(* CODESYS project vertical_levitation_control.library
   TcLibraryId: TE140x Module Vendor|vertical_levitation_control|0.0.0.33
   Company: TE140x Module Vendor
   Title: vertical_levitation_control
   Placeholder: vertical_levitation_control
   Version: 0.0.0.33

Project tree, tasks and I/O mapping:
  POUs/
    function block FB_vertical_levitation_control [ST]: FB_exit, FB_init, nHResult, eInitExceptionHandling, eUpdateExceptionHandling, nExceptionCnt, stActiveException, bInitialized, bExecute
    TcCOM Wrapper/
      function block FB_vertical_levitation_control_TcCOM_InitStruct [ST]: FB_init, FB_afterinit, Reinit, FB_exit, eObjectState, nHResult, ipTcComObject, ipADI, nTaskOid, nTaskPriority, nTaskCycleTimeNs, nTaskPort, nTaskSortOrder, eTraceLevelMax, eModuleCaller, eCallerVerification, eStepSizeAdaptation, eExecutionSequence, bExecute, eAccessLockState, eInitExceptionHandling, eUpdateExceptionHandling, stModuleBuildInfo, bInitialized, nSkippedExecutionCount, stLibraryInfo, stModuleInfo, stModuleGeneratorInfo, stSimulinkModelInfo, evertical_levitation_control_P_Sharing, nvertical_levitation_control_P_Definer, stvertical_levitation_control_P, fSimulationTime, nCycleCount, nExceptionCount, stExceptionInfo
  DUTs/
    data type ST_FB_vertical_levitation_control_FB_Main
    data type ST_FB_vertical_levitation_control_FB_exit
    data type ST_FB_vertical_levitation_control_FB_init
    data type ST_GetSet_HRESULT
    data type E_FpExcptCtrlSetEx
    data type ST_GetSet_E_FpExcptCtrlSetEx
    data type ST_GetSet_ULINT
    data type ST_ExceptionInfo
    data type ST_GetSet_ST_ExceptionInfo
    data type ST_GetSet_BOOL
    data type T_matrix3xdouble
    data type T_matrix2xdouble
    data type T_matrix4xdouble
    data type E_SimTimeStep
    data type E_SolverMode
    data type E_ssMatrixType
    data type ST_RTWRTModelMethodsInfo
    data type E_slJmBdControl
    data type ST_ssSolverInfo
    data type T_matrix8xdouble
    data type T_matrix5xdouble
    data type T_matrix4xlogical
    data type T_matrix8xlogical
    data type ST_B_forcecurrent_BL_vertical_levitation_control_T
    data type ST_B_MATLABFunction_vertical_levitation_control_T
    data type ST_B_vertical_levitation_control_T
    data type T_ZCSigState
    data type T_matrix4xZCSigState
    data type ST_PrevZCX_vertical_levitation_control_T
    data type ST_X_vertical_levitation_control_T
    data type ST_ExtU_vertical_levitation_control_T
    data type ST_ExtY_vertical_levitation_control_T
    data type T_matrix4xbool
    data type ST_XDis_vertical_levitation_control_T
    data type T_matrix22xdouble
    data type T_matrix22x4xdouble
    data type PLREAL
    data type T_matrix4xdoublepointer
    data type ST_ODE4_IntgData
    data type ST_DW_vertical_levitation_control_T
    data type ST_x08a7a7bbd0e5d629f7d70ceec84eacfe
    data type ST_xf09845edab6c83520d8d57def6d6fe1c
    data type ST_RT_MODEL_vertical_levitation_control_T
    data type T_matrix53xdouble
    data type T_matrix1007xdouble
    data type T_matrix19xdouble
    data type T_matrix380xdouble
    data type T_matrix3xlogical
    data type ST_P_vertical_levitation_control_T
    data type E_ModuleCaller
    data type E_CallerVerification
    data type E_StepSizeAdaptation
    data type E_ExecutionSequence1
    data type E_FpExcptCtrlSet
    data type ST_TcMatSim_ModuleGeneratorInfo
    data type ST_TcMatSim_SimulinkModelInfo
    data type E_ParameterSharingType
    data type ST_FB_vertical_levitation_control_TcCOM_InitStruct
    data type ST_FB_vertical_levitation_control_TcCOM_InitStruct_FB_init
    data type ST_FB_vertical_levitation_control_TcCOM_InitStruct_FB_afterinit
    data type ST_FB_vertical_levitation_control_TcCOM_InitStruct_Reinit
    data type ST_FB_vertical_levitation_control_TcCOM_InitStruct_FB_Main
    data type ST_FB_vertical_levitation_control_TcCOM_InitStruct_FB_exit
    data type ST_GetSet_TCOM_STATE
    data type ST_GetSet_ITComObject
    data type ST_GetSet_ITcADI
    data type ST_vertical_levitation_control_U_T
    data type ST_vertical_levitation_control_Y_T
    data type ST_vertical_levitation_control_X_T
    data type ST_vertical_levitation_control_DW_T
    data type ST_GetSet_OTCID
    data type ST_GetSet_UDINT
    data type ST_GetSet_UINT
    data type ST_GetSet_TcTraceLevel
    data type ST_GetSet_E_ModuleCaller
    data type ST_GetSet_E_CallerVerification
    data type ST_GetSet_E_StepSizeAdaptation
    data type ST_GetSet_E_ExecutionSequence1
    data type ST_GetSet_E_FpExcptCtrlSet
    data type ST_ModuleBuildInfo
    data type ST_GetSet_ST_ModuleBuildInfo
    data type ST_LibraryInfo
    data type ST_GetSet_ST_LibraryInfo
    data type ST_ModuleInfo
    data type ST_GetSet_ST_ModuleInfo
    data type ST_GetSet_ST_TcMatSim_ModuleGeneratorInfo
    data type ST_GetSet_ST_TcMatSim_SimulinkModelInfo
    data type ST_GetSet_E_ParameterSharingType
    data type ST_GetSet_ST_P_vertical_levitation_control_T
    data type ST_GetSet_LREAL
  Version/
    global variables Global_Version
*)

// DUTs/ST_FB_vertical_levitation_control_FB_Main
{attribute 'TcIecLibraryType'}
{attribute 'hide'}
TYPE ST_FB_vertical_levitation_control_FB_Main : 
	STRUCT
		{attribute 'GUID' := '18071995-0000-0000-0000-000000000018'}
		pInst : PVOID;
		result : BOOL;
		 {attribute 'hide'}
		_reserved1 : UINT_24_56;
	END_STRUCT
END_TYPE

// DUTs/ST_FB_vertical_levitation_control_FB_exit
{attribute 'TcIecLibraryType'}
{attribute 'hide'}
TYPE ST_FB_vertical_levitation_control_FB_exit : 
	STRUCT
		{attribute 'GUID' := '18071995-0000-0000-0000-000000000018'}
		pInst : PVOID;
		bInCopyCode : BOOL;
		result : BOOL;
		 {attribute 'hide'}
		_reserved1 : UINT_16_48;
	END_STRUCT
END_TYPE

// DUTs/ST_FB_vertical_levitation_control_FB_init
{attribute 'TcIecLibraryType'}
{attribute 'hide'}
TYPE ST_FB_vertical_levitation_control_FB_init : 
	STRUCT
		{attribute 'GUID' := '18071995-0000-0000-0000-000000000018'}
		pInst : PVOID;
		bInitRetains : BOOL;
		bInCopyCode : BOOL;
		result : BOOL;
		 {attribute 'hide'}
		_reserved1 : UINT_8_40;
	END_STRUCT
END_TYPE

// DUTs/ST_GetSet_HRESULT
{attribute 'TcIecLibraryType'}
{attribute 'hide'}
TYPE ST_GetSet_HRESULT : 
	STRUCT
		{attribute 'GUID' := '18071995-0000-0000-0000-000000000018'}
		pInst : PVOID;
		{attribute 'GUID' := '18071995-0000-0000-0000-000000000019'}
		nParam : HRESULT;
		 {attribute 'hide'}
		_reserved1 : UINT_0_32;
	END_STRUCT
END_TYPE

// DUTs/E_FpExcptCtrlSetEx
(* Generated from type 'TcMgSdk.FpExcptCtrlSetEx' *)
{attribute 'TcIecLibraryType'}
TYPE E_FpExcptCtrlSetEx : (
	CallerExceptions:=1, 	(* Use the floating point exception settings provided by the caller *)
	ThrowExceptions:=3, 	(* Enable floating point exceptions on invalid operations and divisions by zero *)
	SuppressExceptions:=13, 	(* Disable floating point exceptions. *)
	LogExceptions:=19, 	(* Log exception information. *)
	LogAndHold:=51, 	(* Log exception information and puase execution of the cyclic code after completion of the actual cycle *)
	LogAndCatch:=83, 	(* Log exception information and immediately terminate execution of the cyclic code. Reinitialization is required to restart. *)
	LogAndDump:=147, 	(* Log exception information, create a dump file with detailed exception information and try to continue execution of the cyclic code *)
	LogHoldAndDump:=179, 	(* Log exception information, create a dump file with detailed exception information and puase execution of the cyclic code after completion of the actual cycle *)
	LogCatchAndDump:=211	(* Log exception information, create a dump file with detailed exception information and immediately terminate execution of the cyclic code. Reinitialization is required to restart. *)
) USINT;
END_TYPE

// DUTs/ST_GetSet_E_FpExcptCtrlSetEx
{attribute 'TcIecLibraryType'}
{attribute 'hide'}
TYPE ST_GetSet_E_FpExcptCtrlSetEx : 
	STRUCT
		{attribute 'GUID' := '18071995-0000-0000-0000-000000000018'}
		pInst : PVOID;
		eParam : E_FpExcptCtrlSetEx;
		 {attribute 'hide'}
		_reserved1 : UINT_24_56;
	END_STRUCT
END_TYPE

// DUTs/ST_GetSet_ULINT
{attribute 'TcIecLibraryType'}
{attribute 'hide'}
TYPE ST_GetSet_ULINT : 
	STRUCT
		{attribute 'GUID' := '18071995-0000-0000-0000-000000000018'}
		pInst : PVOID;
		nParam : ULINT;
	END_STRUCT
END_TYPE

// DUTs/ST_ExceptionInfo
(* Generated from type 'TcMgSdk.ExceptionInfo' *)
{attribute 'TcIecLibraryType'}
TYPE ST_ExceptionInfo : 
	STRUCT
		(* Generated from item 'ExceptionCode' *)
		nExceptionCode : DINT;
		(* Generated from item 'TmxName' *)
		{attribute 'GUID' := '18071995-0000-0000-0000-00010000007F'}
		sTmxName : STRING(127);
		(* Generated from item 'TmxVersion' *)
		nTmxVersion : ARRAY [0..3] OF UDINT;
		(* Generated from item 'InstructionAddr' *)
		nInstructionAddr : UDINT;
		(* Generated from item 'ReturnAddr' *)
		nReturnAddr : ARRAY [0..3] OF UDINT;
		(* Generated from item 'DumpCreated' *)
		bDumpCreated : BOOL;
		 {attribute 'hide'}
		_reserved1 : ARRAY [1..3] OF USINT;
	END_STRUCT
END_TYPE

// DUTs/ST_GetSet_ST_ExceptionInfo
{attribute 'TcIecLibraryType'}
{attribute 'hide'}
TYPE ST_GetSet_ST_ExceptionInfo : 
	STRUCT
		{attribute 'GUID' := '18071995-0000-0000-0000-000000000018'}
		pInst : PVOID;
		stParam : ST_ExceptionInfo;
		 {attribute 'hide'}
		_reserved1 : UINT_0_32;
	END_STRUCT
END_TYPE

// DUTs/ST_GetSet_BOOL
{attribute 'TcIecLibraryType'}
{attribute 'hide'}
TYPE ST_GetSet_BOOL : 
	STRUCT
		{attribute 'GUID' := '18071995-0000-0000-0000-000000000018'}
		pInst : PVOID;
		bParam : BOOL;
		 {attribute 'hide'}
		_reserved1 : UINT_24_56;
	END_STRUCT
END_TYPE

// DUTs/T_matrix3xdouble
(* Generated from type 'matrix3xdouble' *)
{attribute 'TcIecLibraryType'}
TYPE T_matrix3xdouble : ARRAY [0..2] OF LREAL;
END_TYPE

// DUTs/T_matrix2xdouble
(* Generated from type 'matrix2xdouble' *)
{attribute 'TcIecLibraryType'}
TYPE T_matrix2xdouble : ARRAY [0..1] OF LREAL;
END_TYPE

// DUTs/T_matrix4xdouble
(* Generated from type 'matrix4xdouble' *)
{attribute 'TcIecLibraryType'}
TYPE T_matrix4xdouble : ARRAY [0..3] OF LREAL;
END_TYPE

// DUTs/E_SimTimeStep
(* Generated from type 'SimTimeStep' *)
{attribute 'TcIecLibraryType'}
{attribute 'qualified_only' := 'true'}
TYPE E_SimTimeStep : (MINOR_TIME_STEP:=0, MAJOR_TIME_STEP:=1) DINT;
END_TYPE

// DUTs/E_SolverMode
(* Generated from type 'SolverMode' *)
{attribute 'TcIecLibraryType'}
{attribute 'qualified_only' := 'true'}
TYPE E_SolverMode : (SOLVER_MODE_AUTO:=0, SOLVER_MODE_SINGLETASKING:=1, SOLVER_MODE_MULTITASKING:=2) DINT;
END_TYPE

// DUTs/E_ssMatrixType
(* Generated from type 'ssMatrixType' *)
{attribute 'TcIecLibraryType'}
{attribute 'qualified_only' := 'true'}
TYPE E_ssMatrixType : (SS_MATRIX_NONE:=0, SS_MATRIX_CONSTANT:=1, SS_MATRIX_TIMEDEP:=2, SS_MATRIX_STATEDEP:=3) DINT;
END_TYPE

// DUTs/ST_RTWRTModelMethodsInfo
(* Generated from type 'RTWRTModelMethodsInfo' *)
{attribute 'TcIecLibraryType'}
TYPE ST_RTWRTModelMethodsInfo : 
	STRUCT
		(* Generated from item 'rtModelPtr' *)
		{attribute 'GUID' := '18071995-0000-0000-0000-000000000018'}
		prtModelPtr : PVOID;
		(* Generated from item 'rtmInitSizesFcn' *)
		{attribute 'GUID' := '18071995-0000-0000-0000-000000000018'}
		prtmInitSizesFcn : PVOID;
		(* Generated from item 'rtmInitSampTimesFcn' *)
		{attribute 'GUID' := '18071995-0000-0000-0000-000000000018'}
		prtmInitSampTimesFcn : PVOID;
		(* Generated from item 'rtmStartFcn' *)
		{attribute 'GUID' := '18071995-0000-0000-0000-000000000018'}
		prtmStartFcn : PVOID;
		(* Generated from item 'rtmOutputsFcn' *)
		{attribute 'GUID' := '18071995-0000-0000-0000-000000000018'}
		prtmOutputsFcn : PVOID;
		(* Generated from item 'rtmUpdateFcn' *)
		{attribute 'GUID' := '18071995-0000-0000-0000-000000000018'}
		prtmUpdateFcn : PVOID;
		(* Generated from item 'rtmDervisFcn' *)
		{attribute 'GUID' := '18071995-0000-0000-0000-000000000018'}
		prtmDervisFcn : PVOID;
		(* Generated from item 'rtmProjectionFcn' *)
		{attribute 'GUID' := '18071995-0000-0000-0000-000000000018'}
		prtmProjectionFcn : PVOID;
		(* Generated from item 'rtmMassMatrixFcn' *)
		{attribute 'GUID' := '18071995-0000-0000-0000-000000000018'}
		prtmMassMatrixFcn : PVOID;
		(* Generated from item 'rtmForcingFunctionFcn' *)
		{attribute 'GUID' := '18071995-0000-0000-0000-000000000018'}
		prtmForcingFunctionFcn : PVOID;
		(* Generated from item 'rtmTerminateFcn' *)
		{attribute 'GUID' := '18071995-0000-0000-0000-000000000018'}
		prtmTerminateFcn : PVOID;
		(* Generated from item 'rtmDiscreteEventsFcn' *)
		{attribute 'GUID' := '18071995-0000-0000-0000-000000000018'}
		prtmDiscreteEventsFcn : PVOID;
	END_STRUCT
END_TYPE

// DUTs/E_slJmBdControl
(* Generated from type 'slJmBdControl' *)
{attribute 'TcIecLibraryType'}
{attribute 'qualified_only' := 'true'}
TYPE E_slJmBdControl : (SL_JM_BD_AUTO:=0, SL_JM_BD_SPARSE_PERTURBATION:=1, SL_JM_BD_FULL_PERTURBATION:=2, SL_JM_BD_SPARSE_ANALYTICAL:=3, SL_JM_BD_FULL_ANALYTICAL:=4) DINT;
END_TYPE

// DUTs/ST_ssSolverInfo
(* Generated from type 'ssSolverInfo' *)
{attribute 'TcIecLibraryType'}
TYPE ST_ssSolverInfo : 
	STRUCT
		(* Generated from item 'rtModelPtr' *)
		{attribute 'GUID' := '18071995-0000-0000-0000-000000000018'}
		prtModelPtr : PVOID;
		simTimeStepPtr : POINTER TO E_SimTimeStep;
		(* Generated from item 'solverData' *)
		{attribute 'GUID' := '18071995-0000-0000-0000-000000000018'}
		psolverData : PVOID;
		solverName : POINTER TO SINT;
		(* Generated from item 'isVariableStepSolver' *)
		bisVariableStepSolver : BOOL;
		(* Generated from item 'solverNeedsReset' *)
		bsolverNeedsReset : BOOL;
		 {attribute 'hide'}
		_reserved1 : UINT;
		(* Generated from item 'solverMode' *)
		esolverMode : E_SolverMode;
		(* Generated from item 'solverStopTime' *)
		fsolverStopTime : LREAL;
		stepSizePtr : POINTER TO LREAL;
		(* Generated from item 'minStepSize' *)
		fminStepSize : LREAL;
		(* Generated from item 'maxStepSize' *)
		fmaxStepSize : LREAL;
		(* Generated from item 'fixedStepSize' *)
		ffixedStepSize : LREAL;
		(* Generated from item 'solverShapePreserveControl' *)
		nsolverShapePreserveControl : DINT;
		(* Generated from item 'solverMaxConsecutiveMinStep' *)
		nsolverMaxConsecutiveMinStep : DINT;
		(* Generated from item 'maxNumMinSteps' *)
		nmaxNumMinSteps : DINT;
		(* Generated from item 'solverMaxOrder' *)
		nsolverMaxOrder : DINT;
		(* Generated from item 'solverConsecutiveZCsStepRelTol' *)
		fsolverConsecutiveZCsStepRelTol : LREAL;
		(* Generated from item 'solverMaxConsecutiveZCs' *)
		nsolverMaxConsecutiveZCs : DINT;
		(* Generated from item 'solverExtrapolationOrder' *)
		nsolverExtrapolationOrder : DINT;
		(* Generated from item 'solverNumberNewtonIterations' *)
		nsolverNumberNewtonIterations : DINT;
		(* Generated from item 'solverRefineFactor' *)
		nsolverRefineFactor : DINT;
		(* Generated from item 'solverRelTol' *)
		fsolverRelTol : LREAL;
		(* Generated from item 'unused_real_T_1' *)
		funused_real_T_1 : LREAL;
		dXPtr : POINTER TO POINTER TO LREAL;
		tPtr : POINTER TO POINTER TO LREAL;
		numContStatesPtr : POINTER TO DINT;
		contStatesPtr : POINTER TO POINTER TO LREAL;
		numPeriodicContStatesPtr : POINTER TO DINT;
		periodicContStateIndicesPtr : POINTER TO POINTER TO DINT;
		periodicContStateRangesPtr : POINTER TO POINTER TO LREAL;
		zcSignalVector : POINTER TO LREAL;
		zcEventsVector : POINTER TO USINT;
		zcSignalAttrib : POINTER TO USINT;
		(* Generated from item 'zcSignalVectorLength' *)
		nzcSignalVectorLength : DINT;
		 {attribute 'hide'}
		_reserved2 : UINT_0_32;
		reserved : POINTER TO USINT;
		(* Generated from item 'foundContZcEvents' *)
		bfoundContZcEvents : BOOL;
		(* Generated from item 'isAtLeftPostOfContZcEvent' *)
		bisAtLeftPostOfContZcEvent : BOOL;
		(* Generated from item 'isAtRightPostOfContZcEvent' *)
		bisAtRightPostOfContZcEvent : BOOL;
		(* Generated from item 'adaptiveZcDetection' *)
		badaptiveZcDetection : BOOL;
		(* Generated from item 'numZcSignals' *)
		nnumZcSignals : DINT;
		(* Generated from item 'stateProjection' *)
		bstateProjection : BOOL;
		(* Generated from item 'robustResetMethod' *)
		brobustResetMethod : BOOL;
		(* Generated from item 'updateJacobianAtReset' *)
		bupdateJacobianAtReset : BOOL;
		(* Generated from item 'consistencyChecking' *)
		bconsistencyChecking : BOOL;
		(* Generated from item 'massMatrixType' *)
		emassMatrixType : E_ssMatrixType;
		(* Generated from item 'massMatrixNzMax' *)
		nmassMatrixNzMax : DINT;
		 {attribute 'hide'}
		_reserved3 : UINT_0_32;
		massMatrixIr : POINTER TO DINT;
		massMatrixJc : POINTER TO DINT;
		massMatrixPr : POINTER TO LREAL;
		errStatusPtr : POINTER TO POINTER TO SINT;
		modelMethodsPtr : POINTER TO ST_RTWRTModelMethodsInfo;
		(* Generated from item 'zcThreshold' *)
		fzcThreshold : LREAL;
		(* Generated from item 'reserved_1' *)
		nreserved_1 : DINT;
		(* Generated from item 'consecutiveZCsError' *)
		nconsecutiveZCsError : DINT;
		(* Generated from item 'CTOutputIncnstWithState' *)
		bCTOutputIncnstWithState : BOOL;
		(* Generated from item 'isComputingJacobian' *)
		bisComputingJacobian : BOOL;
		 {attribute 'hide'}
		_reserved4 : UINT;
		(* Generated from item 'solverJacobianMethodControl' *)
		esolverJacobianMethodControl : E_slJmBdControl;
		(* Generated from item 'ignoredZcDiagnostic' *)
		nignoredZcDiagnostic : DINT;
		(* Generated from item 'maskedZcDiagnostic' *)
		nmaskedZcDiagnostic : DINT;
		(* Generated from item 'isOutputMethodComputed' *)
		bisOutputMethodComputed : BOOL;
		 {attribute 'hide'}
		_reserved5 : ARRAY [1..3] OF USINT;
		(* Generated from item 'maxZcBracketingIterations' *)
		nmaxZcBracketingIterations : DINT;
		(* Generated from item 'isMinorTimeStepWithModeChange' *)
		bisMinorTimeStepWithModeChange : BOOL;
		 {attribute 'hide'}
		_reserved6 : ARRAY [1..3] OF USINT;
		(* Generated from item 'maxZcPerStep' *)
		nmaxZcPerStep : DINT;
		zcSignalPtr : POINTER TO POINTER TO LREAL;
		(* Generated from item 'contStateDisabledPtr' *)
		bcontStateDisabledPtr : POINTER TO POINTER TO BOOL;
		(* Generated from item 'isContModeFrozen' *)
		bisContModeFrozen : BOOL;
		 {attribute 'hide'}
		_reserved7 : ARRAY [1..7] OF USINT;
	END_STRUCT
END_TYPE

// DUTs/T_matrix8xdouble
(* Generated from type 'matrix8xdouble' *)
{attribute 'TcIecLibraryType'}
TYPE T_matrix8xdouble : ARRAY [0..7] OF LREAL;
END_TYPE

// DUTs/T_matrix5xdouble
(* Generated from type 'matrix5xdouble' *)
{attribute 'TcIecLibraryType'}
TYPE T_matrix5xdouble : ARRAY [0..4] OF LREAL;
END_TYPE

// DUTs/T_matrix4xlogical
(* Generated from type 'matrix4xlogical' *)
{attribute 'TcIecLibraryType'}
{attribute 'BaseTypeGUID' := '18071995-0000-0000-0000-000000000030'}
TYPE T_matrix4xlogical : ARRAY [0..3] OF BOOL;
END_TYPE

// DUTs/T_matrix8xlogical
(* Generated from type 'matrix8xlogical' *)
{attribute 'TcIecLibraryType'}
{attribute 'BaseTypeGUID' := '18071995-0000-0000-0000-000000000030'}
TYPE T_matrix8xlogical : ARRAY [0..7] OF BOOL;
END_TYPE

// DUTs/ST_B_forcecurrent_BL_vertical_levitation_control_T
(* Generated from type 'B_forcecurrent_BL_vertical_levitation_control_T' *)
{attribute 'TcIecLibraryType'}
TYPE ST_B_forcecurrent_BL_vertical_levitation_control_T : 
	STRUCT
		(* Generated from item 'current_reqf' *)
		fcurrent_reqf : LREAL;
		(* Generated from item 'current_reqb' *)
		fcurrent_reqb : LREAL;
	END_STRUCT
END_TYPE

// DUTs/ST_B_MATLABFunction_vertical_levitation_control_T
(* Generated from type 'B_MATLABFunction_vertical_levitation_control_T' *)
{attribute 'TcIecLibraryType'}
TYPE ST_B_MATLABFunction_vertical_levitation_control_T : 
	STRUCT
		(* Generated from item 'y' *)
		ay : T_matrix8xdouble;
	END_STRUCT
END_TYPE

// DUTs/ST_B_vertical_levitation_control_T
(* Generated from type 'B_vertical_levitation_control_T' *)
{attribute 'TcIecLibraryType'}
TYPE ST_B_vertical_levitation_control_T : 
	STRUCT
		(* Generated from item 'UnitDelay' *)
		aUnitDelay : T_matrix4xdouble;
		(* Generated from item 'Switch1' *)
		aSwitch1 : T_matrix4xdouble;
		(* Generated from item 'Switch1_d' *)
		aSwitch1_d : T_matrix4xdouble;
		(* Generated from item 'Gain3' *)
		fGain3 : LREAL;
		(* Generated from item 'Gain7' *)
		fGain7 : LREAL;
		(* Generated from item 'Switch2' *)
		aSwitch2 : T_matrix4xdouble;
		(* Generated from item 'select_maxs' *)
		aselect_maxs : T_matrix4xdouble;
		(* Generated from item 'Delay' *)
		aDelay : T_matrix3xdouble;
		(* Generated from item 'UnitDelay1' *)
		fUnitDelay1 : LREAL;
		(* Generated from item 'FilterCoefficient' *)
		fFilterCoefficient : LREAL;
		(* Generated from item 'Saturation' *)
		fSaturation : LREAL;
		(* Generated from item 'error_integrator' *)
		ferror_integrator : LREAL;
		(* Generated from item 'Gain10' *)
		fGain10 : LREAL;
		(* Generated from item 'Integrator' *)
		fIntegrator : LREAL;
		(* Generated from item 'Filtertotgain' *)
		fFiltertotgain : LREAL;
		(* Generated from item 'Add4' *)
		fAdd4 : LREAL;
		(* Generated from item 'UnitDelay1_g' *)
		fUnitDelay1_g : LREAL;
		(* Generated from item 'Sum' *)
		fSum : LREAL;
		(* Generated from item 'Gain12' *)
		fGain12 : LREAL;
		(* Generated from item 'Integrator_g' *)
		fIntegrator_g : LREAL;
		(* Generated from item 'K_D_roll' *)
		fK_D_roll : LREAL;
		(* Generated from item 'Filterrollgain' *)
		fFilterrollgain : LREAL;
		(* Generated from item 'TSamp' *)
		fTSamp : LREAL;
		(* Generated from item 'Diff' *)
		fDiff : LREAL;
		(* Generated from item 'Add4_g' *)
		fAdd4_g : LREAL;
		(* Generated from item 'UnitDelay1_i' *)
		fUnitDelay1_i : LREAL;
		(* Generated from item 'Add4_gu' *)
		fAdd4_gu : LREAL;
		(* Generated from item 'UnitDelay1_d' *)
		fUnitDelay1_d : LREAL;
		(* Generated from item 'Switch' *)
		fSwitch : LREAL;
		(* Generated from item 'Gain13' *)
		fGain13 : LREAL;
		(* Generated from item 'Integrator_i' *)
		fIntegrator_i : LREAL;
		(* Generated from item 'Filterpitgain' *)
		fFilterpitgain : LREAL;
		(* Generated from item 'Add4_l' *)
		fAdd4_l : LREAL;
		(* Generated from item 'UnitDelay1_e' *)
		fUnitDelay1_e : LREAL;
		(* Generated from item 'Sum_j' *)
		fSum_j : LREAL;
		(* Generated from item 'select_mins' *)
		aselect_mins : T_matrix4xdouble;
		(* Generated from item 'Switch_i' *)
		fSwitch_i : LREAL;
		(* Generated from item 'UnitDelay1_m' *)
		fUnitDelay1_m : LREAL;
		(* Generated from item 'FilterCoefficient_l' *)
		fFilterCoefficient_l : LREAL;
		(* Generated from item 'Saturation_p' *)
		fSaturation_p : LREAL;
		(* Generated from item 'Switch1_a' *)
		fSwitch1_a : LREAL;
		(* Generated from item 'UnitDelay1_n' *)
		fUnitDelay1_n : LREAL;
		(* Generated from item 'FilterCoefficient_o' *)
		fFilterCoefficient_o : LREAL;
		(* Generated from item 'Saturation_pi' *)
		fSaturation_pi : LREAL;
		(* Generated from item 'Switch2_j' *)
		fSwitch2_j : LREAL;
		(* Generated from item 'F_hemsfinal' *)
		aF_hemsfinal : T_matrix4xdouble;
		(* Generated from item 'Switch2_f' *)
		aSwitch2_f : T_matrix8xdouble;
		(* Generated from item 'Switch_o' *)
		fSwitch_o : LREAL;
		(* Generated from item 'Switch_j' *)
		fSwitch_j : LREAL;
		(* Generated from item 'Switch_k' *)
		fSwitch_k : LREAL;
		(* Generated from item 'Divide' *)
		fDivide : LREAL;
		(* Generated from item 'Add5' *)
		fAdd5 : LREAL;
		(* Generated from item 'Add6' *)
		fAdd6 : LREAL;
		(* Generated from item 'Gain' *)
		fGain : LREAL;
		(* Generated from item 'UnitDelay2' *)
		fUnitDelay2 : LREAL;
		(* Generated from item 'Sum4' *)
		fSum4 : LREAL;
		(* Generated from item 'Sum5' *)
		fSum5 : LREAL;
		(* Generated from item 'Add5_p' *)
		fAdd5_p : LREAL;
		(* Generated from item 'Add6_l' *)
		fAdd6_l : LREAL;
		(* Generated from item 'Gain_m' *)
		fGain_m : LREAL;
		(* Generated from item 'UnitDelay2_i' *)
		fUnitDelay2_i : LREAL;
		(* Generated from item 'Sum4_d' *)
		fSum4_d : LREAL;
		(* Generated from item 'Sum5_m' *)
		fSum5_m : LREAL;
		(* Generated from item 'Add5_f' *)
		fAdd5_f : LREAL;
		(* Generated from item 'Add6_a' *)
		fAdd6_a : LREAL;
		(* Generated from item 'Gain_j' *)
		fGain_j : LREAL;
		(* Generated from item 'UnitDelay2_m' *)
		fUnitDelay2_m : LREAL;
		(* Generated from item 'Sum4_g' *)
		fSum4_g : LREAL;
		(* Generated from item 'Sum5_g' *)
		fSum5_g : LREAL;
		(* Generated from item 'Add5_h' *)
		fAdd5_h : LREAL;
		(* Generated from item 'Add6_h' *)
		fAdd6_h : LREAL;
		(* Generated from item 'Gain_l' *)
		fGain_l : LREAL;
		(* Generated from item 'UnitDelay2_o' *)
		fUnitDelay2_o : LREAL;
		(* Generated from item 'Sum4_i' *)
		fSum4_i : LREAL;
		(* Generated from item 'Sum5_j' *)
		fSum5_j : LREAL;
		(* Generated from item 'IsPeak1' *)
		aIsPeak1 : T_matrix4xdouble;
		(* Generated from item 'Switch2_d' *)
		aSwitch2_d : T_matrix4xdouble;
		(* Generated from item 'F_netpostfm' *)
		aF_netpostfm : T_matrix3xdouble;
		(* Generated from item 'clamppit' *)
		fclamppit : LREAL;
		(* Generated from item 'clamproll' *)
		fclamproll : LREAL;
		(* Generated from item 'clamptot' *)
		fclamptot : LREAL;
		(* Generated from item 'K_I_tot' *)
		fK_I_tot : LREAL;
		(* Generated from item 'K_I_roll' *)
		fK_I_roll : LREAL;
		(* Generated from item 'K_I_pit' *)
		fK_I_pit : LREAL;
		(* Generated from item 'current_reqf' *)
		fcurrent_reqf : LREAL;
		(* Generated from item 'current_reqb' *)
		fcurrent_reqb : LREAL;
		(* Generated from item 'current_reqf_c' *)
		fcurrent_reqf_c : LREAL;
		(* Generated from item 'current_reqb_c' *)
		fcurrent_reqb_c : LREAL;
		(* Generated from item 'F_hems' *)
		aF_hems : T_matrix4xdouble;
		(* Generated from item 'Switch2_l' *)
		aSwitch2_l : T_matrix4xdouble;
		(* Generated from item 'Sum5_f' *)
		fSum5_f : LREAL;
		(* Generated from item 'Is' *)
		aIs : T_matrix4xdouble;
		(* Generated from item 'satn' *)
		asatn : T_matrix8xdouble;
		(* Generated from item 'airgaps_avg' *)
		aairgaps_avg : T_matrix4xdouble;
		(* Generated from item 'airgap_diff' *)
		fairgap_diff : LREAL;
		(* Generated from item 'tau_x' *)
		ftau_x : LREAL;
		(* Generated from item 'Sum_l' *)
		fSum_l : LREAL;
		(* Generated from item 'corrected_out' *)
		fcorrected_out : LREAL;
		(* Generated from item 'corrected_out_j' *)
		fcorrected_out_j : LREAL;
		(* Generated from item 'corrected_out_o' *)
		fcorrected_out_o : LREAL;
		(* Generated from item 'F_hems_b' *)
		aF_hems_b : T_matrix4xdouble;
		(* Generated from item 'clamp_tot' *)
		aclamp_tot : T_matrix2xdouble;
		(* Generated from item 'clamp_roll' *)
		aclamp_roll : T_matrix2xdouble;
		(* Generated from item 'clamp_pit' *)
		aclamp_pit : T_matrix2xdouble;
		(* Generated from item 'counter' *)
		acounter : T_matrix5xdouble;
		(* Generated from item 'F_dof_sat' *)
		aF_dof_sat : T_matrix3xdouble;
		(* Generated from item 'sat_fail' *)
		fsat_fail : LREAL;
		(* Generated from item 'q' *)
		fq : LREAL;
		(* Generated from item 'q_m' *)
		fq_m : LREAL;
		(* Generated from item 'q_f' *)
		fq_f : LREAL;
		(* Generated from item 'q_d' *)
		fq_d : LREAL;
		(* Generated from item 'UnaryMinus' *)
		fUnaryMinus : LREAL;
		(* Generated from item 'UnaryMinus_b' *)
		fUnaryMinus_b : LREAL;
		(* Generated from item 'UnaryMinus_n' *)
		fUnaryMinus_n : LREAL;
		(* Generated from item 'UnaryMinus_l' *)
		fUnaryMinus_l : LREAL;
		(* Generated from item 'Integrator2' *)
		aIntegrator2 : T_matrix4xdouble;
		(* Generated from item 'Switch_ka' *)
		aSwitch_ka : T_matrix4xdouble;
		(* Generated from item 'K_P_tot' *)
		fK_P_tot : LREAL;
		(* Generated from item 'Product1' *)
		fProduct1 : LREAL;
		(* Generated from item 'Product1_p' *)
		fProduct1_p : LREAL;
		(* Generated from item 'Product1_i' *)
		fProduct1_i : LREAL;
		(* Generated from item 'TmpSignalConversionAtSFunctionInport1' *)
		aTmpSignalConversionAtSFunctionInport1 : T_matrix3xdouble;
		(* Generated from item 't' *)
		ft : LREAL;
		(* Generated from item 's' *)
		fs : LREAL;
		(* Generated from item 'v' *)
		fv : LREAL;
		(* Generated from item 't_m' *)
		ft_m : LREAL;
		(* Generated from item 's_b' *)
		fs_b : LREAL;
		(* Generated from item 'v_i' *)
		fv_i : LREAL;
		(* Generated from item 't_k' *)
		ft_k : LREAL;
		(* Generated from item 's_i' *)
		fs_i : LREAL;
		(* Generated from item 'v_l' *)
		fv_l : LREAL;
		(* Generated from item 't_i' *)
		ft_i : LREAL;
		(* Generated from item 's_iy' *)
		fs_iy : LREAL;
		(* Generated from item 'v_if' *)
		fv_if : LREAL;
		(* Generated from item 'Integrator_f' *)
		fIntegrator_f : LREAL;
		(* Generated from item 'Switch_h' *)
		fSwitch_h : LREAL;
		(* Generated from item 'u' *)
		fu : LREAL;
		(* Generated from item 'u_h' *)
		fu_h : LREAL;
		(* Generated from item 'u_ha' *)
		fu_ha : LREAL;
		(* Generated from item 'Final_ON' *)
		aFinal_ON : T_matrix8xdouble;
		(* Generated from item 'Abs1' *)
		aAbs1 : T_matrix4xdouble;
		(* Generated from item 'IntegralGain' *)
		fIntegralGain : LREAL;
		(* Generated from item 'u_f' *)
		fu_f : LREAL;
		(* Generated from item 'IntegralGain_e' *)
		fIntegralGain_e : LREAL;
		(* Generated from item 'SignPreSat' *)
		fSignPreSat : LREAL;
		(* Generated from item 'IntegralGain_h' *)
		fIntegralGain_h : LREAL;
		(* Generated from item 'Product4' *)
		fProduct4 : LREAL;
		(* Generated from item 'Product4_b' *)
		fProduct4_b : LREAL;
		(* Generated from item 'Product4_e' *)
		fProduct4_e : LREAL;
		(* Generated from item 'Product4_d' *)
		fProduct4_d : LREAL;
		(* Generated from item 'Product3' *)
		fProduct3 : LREAL;
		(* Generated from item 'SignPreSat_g' *)
		fSignPreSat_g : LREAL;
		(* Generated from item 'SignPreSat_b' *)
		fSignPreSat_b : LREAL;
		(* Generated from item 'Product4_a' *)
		fProduct4_a : LREAL;
		(* Generated from item 'Sign' *)
		fSign : LREAL;
		(* Generated from item 'Sign1' *)
		fSign1 : LREAL;
		(* Generated from item 'Delay1' *)
		fDelay1 : REAL;
		(* Generated from item 'fmsatfailordisabled' *)
		ffmsatfailordisabled : REAL;
		(* Generated from item 'hard_disable_fmm' *)
		fhard_disable_fmm : REAL;
		(* Generated from item 'enabled' *)
		nenabled : USINT;
		(* Generated from item 'DataTypeConv2' *)
		nDataTypeConv2 : SINT;
		(* Generated from item 'DataTypeConv1' *)
		nDataTypeConv1 : SINT;
		(* Generated from item 'didfmcausesattofail' *)
		adidfmcausesattofail : T_matrix4xlogical;
		(* Generated from item 'AND3' *)
		bAND3 : BOOL;
		(* Generated from item 'Memory' *)
		bMemory : BOOL;
		(* Generated from item 'AND3_d' *)
		bAND3_d : BOOL;
		(* Generated from item 'Memory_p' *)
		bMemory_p : BOOL;
		(* Generated from item 'AND3_l' *)
		bAND3_l : BOOL;
		(* Generated from item 'Memory_f' *)
		bMemory_f : BOOL;
		(* Generated from item 'y' *)
		_by : BOOL;
		(* Generated from item 'LowerRelop1' *)
		aLowerRelop1 : T_matrix4xlogical;
		(* Generated from item 'UpperRelop' *)
		aUpperRelop : T_matrix4xlogical;
		(* Generated from item 'LowerRelop1_c' *)
		aLowerRelop1_c : T_matrix8xlogical;
		(* Generated from item 'UpperRelop_o' *)
		aUpperRelop_o : T_matrix8xlogical;
		(* Generated from item 'LowerRelop1_e' *)
		aLowerRelop1_e : T_matrix4xlogical;
		(* Generated from item 'CastToBoolean' *)
		bCastToBoolean : BOOL;
		(* Generated from item 'AND' *)
		bAND : BOOL;
		(* Generated from item 'sf_forcecurrent_FR' *)
		stsf_forcecurrent_FR : ST_B_forcecurrent_BL_vertical_levitation_control_T;
		(* Generated from item 'sf_forcecurrent_BL' *)
		stsf_forcecurrent_BL : ST_B_forcecurrent_BL_vertical_levitation_control_T;
		(* Generated from item 'sf_MATLABFunction1' *)
		stsf_MATLABFunction1 : ST_B_MATLABFunction_vertical_levitation_control_T;
		(* Generated from item 'sf_MATLABFunction' *)
		stsf_MATLABFunction : ST_B_MATLABFunction_vertical_levitation_control_T;
	END_STRUCT
END_TYPE

// DUTs/T_ZCSigState
(* Generated from type 'ZCSigState' *)
{attribute 'TcIecLibraryType'}
TYPE T_ZCSigState : USINT;
END_TYPE

// DUTs/T_matrix4xZCSigState
(* Generated from type 'matrix4xZCSigState' *)
{attribute 'TcIecLibraryType'}
{attribute 'BaseTypeGUID' := 'CF0EC509-8CFA-173E-6D32-2A6837BC8565'}
TYPE T_matrix4xZCSigState : ARRAY [0..3] OF T_ZCSigState;
END_TYPE

// DUTs/ST_PrevZCX_vertical_levitation_control_T
(* Generated from type 'PrevZCX_vertical_levitation_control_T' *)
{attribute 'TcIecLibraryType'}
TYPE ST_PrevZCX_vertical_levitation_control_T : 
	STRUCT
		(* Generated from item 'Integrator1_Reset_ZCE' *)
		aIntegrator1_Reset_ZCE : T_matrix4xZCSigState;
		(* Generated from item 'Integrator_Reset_ZCE' *)
		nIntegrator_Reset_ZCE : T_ZCSigState;
		(* Generated from item 'Filter_Reset_ZCE' *)
		nFilter_Reset_ZCE : T_ZCSigState;
		(* Generated from item 'error_integrator_Reset_ZCE' *)
		nerror_integrator_Reset_ZCE : T_ZCSigState;
		(* Generated from item 'time_integrator_Reset_ZCE' *)
		ntime_integrator_Reset_ZCE : T_ZCSigState;
		(* Generated from item 'Integrator_Reset_ZCE_k' *)
		nIntegrator_Reset_ZCE_k : T_ZCSigState;
		(* Generated from item 'Filtertot_Reset_ZCE' *)
		nFiltertot_Reset_ZCE : T_ZCSigState;
		(* Generated from item 'Integrator_Reset_ZCE_m' *)
		nIntegrator_Reset_ZCE_m : T_ZCSigState;
		(* Generated from item 'Filterroll_Reset_ZCE' *)
		nFilterroll_Reset_ZCE : T_ZCSigState;
		(* Generated from item 'Integrator_Reset_ZCE_km' *)
		nIntegrator_Reset_ZCE_km : T_ZCSigState;
		(* Generated from item 'Filterpit_Reset_ZCE' *)
		nFilterpit_Reset_ZCE : T_ZCSigState;
		(* Generated from item 'Integrator_Reset_ZCE_b' *)
		nIntegrator_Reset_ZCE_b : T_ZCSigState;
		(* Generated from item 'Filter_Reset_ZCE_m' *)
		nFilter_Reset_ZCE_m : T_ZCSigState;
		(* Generated from item 'Integrator_Reset_ZCE_d' *)
		nIntegrator_Reset_ZCE_d : T_ZCSigState;
		(* Generated from item 'Filter_Reset_ZCE_a' *)
		nFilter_Reset_ZCE_a : T_ZCSigState;
		(* Generated from item 'Integrator2_Reset_ZCE' *)
		aIntegrator2_Reset_ZCE : T_matrix4xZCSigState;
	END_STRUCT
END_TYPE

// DUTs/ST_X_vertical_levitation_control_T
(* Generated from type 'X_vertical_levitation_control_T' *)
{attribute 'TcIecLibraryType'}
TYPE ST_X_vertical_levitation_control_T : 
	STRUCT
		(* Generated from item 'Integrator1_CSTATE' *)
		aIntegrator1_CSTATE : T_matrix4xdouble;
		(* Generated from item 'Integrator_CSTATE' *)
		fIntegrator_CSTATE : LREAL;
		(* Generated from item 'Filter_CSTATE' *)
		fFilter_CSTATE : LREAL;
		(* Generated from item 'error_integrator_CSTATE' *)
		ferror_integrator_CSTATE : LREAL;
		(* Generated from item 'time_integrator_CSTATE' *)
		ftime_integrator_CSTATE : LREAL;
		(* Generated from item 'Integrator_CSTATE_p' *)
		fIntegrator_CSTATE_p : LREAL;
		(* Generated from item 'Filtertot_CSTATE' *)
		fFiltertot_CSTATE : LREAL;
		(* Generated from item 'Integrator_CSTATE_k' *)
		fIntegrator_CSTATE_k : LREAL;
		(* Generated from item 'Filterroll_CSTATE' *)
		fFilterroll_CSTATE : LREAL;
		(* Generated from item 'Integrator_CSTATE_pl' *)
		fIntegrator_CSTATE_pl : LREAL;
		(* Generated from item 'Filterpit_CSTATE' *)
		fFilterpit_CSTATE : LREAL;
		(* Generated from item 'Integrator_CSTATE_c' *)
		fIntegrator_CSTATE_c : LREAL;
		(* Generated from item 'Filter_CSTATE_j' *)
		fFilter_CSTATE_j : LREAL;
		(* Generated from item 'Integrator_CSTATE_pq' *)
		fIntegrator_CSTATE_pq : LREAL;
		(* Generated from item 'Filter_CSTATE_b' *)
		fFilter_CSTATE_b : LREAL;
		(* Generated from item 'Integrator2_CSTATE' *)
		aIntegrator2_CSTATE : T_matrix4xdouble;
	END_STRUCT
END_TYPE

// DUTs/ST_ExtU_vertical_levitation_control_T
(* Generated from type 'ExtU_vertical_levitation_control_T' *)
{attribute 'TcIecLibraryType'}
TYPE ST_ExtU_vertical_levitation_control_T : 
	STRUCT
		(* Generated from item 'z_avg' *)
		fz_avg : LREAL;
		(* Generated from item 'roll_measured' *)
		froll_measured : LREAL;
		(* Generated from item 'pitch_measured' *)
		fpitch_measured : LREAL;
		(* Generated from item 'ems_roll' *)
		fems_roll : LREAL;
		(* Generated from item 'F_imu' *)
		aF_imu : T_matrix3xdouble;
		(* Generated from item 'gyro_imu' *)
		agyro_imu : T_matrix3xdouble;
		(* Generated from item 'motor_Fy_l' *)
		fmotor_Fy_l : LREAL;
		(* Generated from item 'motor_Fy_r' *)
		fmotor_Fy_r : LREAL;
		(* Generated from item 'Feedback_current_hems' *)
		fFeedback_current_hems : LREAL;
	END_STRUCT
END_TYPE

// DUTs/ST_ExtY_vertical_levitation_control_T
(* Generated from type 'ExtY_vertical_levitation_control_T' *)
{attribute 'TcIecLibraryType'}
TYPE ST_ExtY_vertical_levitation_control_T : 
	STRUCT
		(* Generated from item 'I_VFL' *)
		aI_VFL : T_matrix2xdouble;
		(* Generated from item 'I_VFR' *)
		aI_VFR : T_matrix2xdouble;
		(* Generated from item 'I_VBL' *)
		aI_VBL : T_matrix2xdouble;
		(* Generated from item 'I_VBR' *)
		aI_VBR : T_matrix2xdouble;
		(* Generated from item 'F_hems' *)
		aF_hems : T_matrix4xdouble;
		(* Generated from item 'F_requested' *)
		aF_requested : T_matrix3xdouble;
		(* Generated from item 'integral_terms' *)
		aintegral_terms : T_matrix3xdouble;
		(* Generated from item 'sat_failed' *)
		fsat_failed : LREAL;
		(* Generated from item 'net_post_sat' *)
		anet_post_sat : T_matrix3xdouble;
		(* Generated from item 'z_target_adjusted' *)
		fz_target_adjusted : LREAL;
		(* Generated from item 'Max_allowed_current' *)
		aMax_allowed_current : T_matrix4xdouble;
		(* Generated from item 'Min_allowed_current' *)
		aMin_allowed_current : T_matrix4xdouble;
		(* Generated from item 'Avg_total_hems_current' *)
		fAvg_total_hems_current : LREAL;
		(* Generated from item 'Avg_current_hems' *)
		fAvg_current_hems : LREAL;
	END_STRUCT
END_TYPE

// DUTs/T_matrix4xbool
(* Generated from type 'matrix4xbool' *)
{attribute 'TcIecLibraryType'}
{attribute 'BaseTypeGUID' := '18071995-0000-0000-0000-000000000030'}
TYPE T_matrix4xbool : ARRAY [0..3] OF BOOL;
END_TYPE

// DUTs/ST_XDis_vertical_levitation_control_T
(* Generated from type 'XDis_vertical_levitation_control_T' *)
{attribute 'TcIecLibraryType'}
TYPE ST_XDis_vertical_levitation_control_T : 
	STRUCT
		(* Generated from item 'Integrator1_CSTATE' *)
		aIntegrator1_CSTATE : T_matrix4xbool;
		(* Generated from item 'Integrator_CSTATE' *)
		bIntegrator_CSTATE : BOOL;
		(* Generated from item 'Filter_CSTATE' *)
		bFilter_CSTATE : BOOL;
		(* Generated from item 'error_integrator_CSTATE' *)
		berror_integrator_CSTATE : BOOL;
		(* Generated from item 'time_integrator_CSTATE' *)
		btime_integrator_CSTATE : BOOL;
		(* Generated from item 'Integrator_CSTATE_p' *)
		bIntegrator_CSTATE_p : BOOL;
		(* Generated from item 'Filtertot_CSTATE' *)
		bFiltertot_CSTATE : BOOL;
		(* Generated from item 'Integrator_CSTATE_k' *)
		bIntegrator_CSTATE_k : BOOL;
		(* Generated from item 'Filterroll_CSTATE' *)
		bFilterroll_CSTATE : BOOL;
		(* Generated from item 'Integrator_CSTATE_pl' *)
		bIntegrator_CSTATE_pl : BOOL;
		(* Generated from item 'Filterpit_CSTATE' *)
		bFilterpit_CSTATE : BOOL;
		(* Generated from item 'Integrator_CSTATE_c' *)
		bIntegrator_CSTATE_c : BOOL;
		(* Generated from item 'Filter_CSTATE_j' *)
		bFilter_CSTATE_j : BOOL;
		(* Generated from item 'Integrator_CSTATE_pq' *)
		bIntegrator_CSTATE_pq : BOOL;
		(* Generated from item 'Filter_CSTATE_b' *)
		bFilter_CSTATE_b : BOOL;
		(* Generated from item 'Integrator2_CSTATE' *)
		aIntegrator2_CSTATE : T_matrix4xbool;
	END_STRUCT
END_TYPE

// DUTs/T_matrix22xdouble
(* Generated from type 'matrix22xdouble' *)
{attribute 'TcIecLibraryType'}
TYPE T_matrix22xdouble : ARRAY [0..21] OF LREAL;
END_TYPE

// DUTs/T_matrix22x4xdouble
(* Generated from type 'matrix22x4xdouble' *)
{attribute 'TcIecLibraryType'}
TYPE T_matrix22x4xdouble : ARRAY [0..3,0..21] OF LREAL;
END_TYPE

// DUTs/PLREAL
{attribute 'TcIecLibraryType'}
TYPE PLREAL : POINTER TO LREAL;
END_TYPE

// DUTs/T_matrix4xdoublepointer
(* Generated from type 'matrix4xdouble *' *)
{attribute 'TcIecLibraryType'}
{attribute 'BaseTypeGUID' := '2CE33DB5-EBD3-49F7-1FA0-F8105FFA7B54'}
TYPE T_matrix4xdoublepointer : ARRAY [0..3] OF PLREAL;
END_TYPE

// DUTs/ST_ODE4_IntgData
(* Generated from type 'ODE4_IntgData' *)
{attribute 'TcIecLibraryType'}
{attribute 'pack_mode' := '1'}
TYPE ST_ODE4_IntgData : 
	STRUCT
		y : POINTER TO LREAL;
		(* Generated from item 'f' *)
		af : T_matrix4xdoublepointer;
	END_STRUCT
END_TYPE

// DUTs/ST_DW_vertical_levitation_control_T
(* Generated from type 'DW_vertical_levitation_control_T' *)
{attribute 'TcIecLibraryType'}
TYPE ST_DW_vertical_levitation_control_T : 
	STRUCT
		(* Generated from item 'UnitDelay_DSTATE' *)
		aUnitDelay_DSTATE : T_matrix4xdouble;
		(* Generated from item 'Delay_DSTATE' *)
		aDelay_DSTATE : T_matrix3xdouble;
		(* Generated from item 'UnitDelay1_DSTATE' *)
		fUnitDelay1_DSTATE : LREAL;
		(* Generated from item 'UnitDelay1_DSTATE_a' *)
		fUnitDelay1_DSTATE_a : LREAL;
		(* Generated from item 'UD_DSTATE' *)
		fUD_DSTATE : LREAL;
		(* Generated from item 'UnitDelay1_DSTATE_j' *)
		fUnitDelay1_DSTATE_j : LREAL;
		(* Generated from item 'UnitDelay1_DSTATE_e' *)
		fUnitDelay1_DSTATE_e : LREAL;
		(* Generated from item 'UnitDelay1_DSTATE_ev' *)
		fUnitDelay1_DSTATE_ev : LREAL;
		(* Generated from item 'UnitDelay1_DSTATE_c' *)
		fUnitDelay1_DSTATE_c : LREAL;
		(* Generated from item 'UnitDelay1_DSTATE_d' *)
		fUnitDelay1_DSTATE_d : LREAL;
		(* Generated from item 'UnitDelay2_DSTATE' *)
		fUnitDelay2_DSTATE : LREAL;
		(* Generated from item 'UnitDelay2_DSTATE_l' *)
		fUnitDelay2_DSTATE_l : LREAL;
		(* Generated from item 'UnitDelay2_DSTATE_lt' *)
		fUnitDelay2_DSTATE_lt : LREAL;
		(* Generated from item 'UnitDelay2_DSTATE_j' *)
		fUnitDelay2_DSTATE_j : LREAL;
		(* Generated from item 'Delay1_DSTATE' *)
		fDelay1_DSTATE : REAL;
		(* Generated from item 'Memory_PreviousInput' *)
		bMemory_PreviousInput : BOOL;
		(* Generated from item 'Memory_PreviousInput_l' *)
		bMemory_PreviousInput_l : BOOL;
		(* Generated from item 'Memory_PreviousInput_a' *)
		bMemory_PreviousInput_a : BOOL;
		 {attribute 'hide'}
		_reserved1 : USINT;
	END_STRUCT
END_TYPE

// DUTs/ST_x08a7a7bbd0e5d629f7d70ceec84eacfe
(* Generated from type 'x08a7a7bbd0e5d629f7d70ceec84eacfe' *)
{attribute 'TcIecLibraryType'}
TYPE ST_x08a7a7bbd0e5d629f7d70ceec84eacfe : 
	STRUCT
		(* Generated from item 'numContStates' *)
		nnumContStates : DINT;
		(* Generated from item 'numPeriodicContStates' *)
		nnumPeriodicContStates : DINT;
		(* Generated from item 'numSampTimes' *)
		nnumSampTimes : DINT;
	END_STRUCT
END_TYPE

// DUTs/ST_xf09845edab6c83520d8d57def6d6fe1c
(* Generated from type 'xf09845edab6c83520d8d57def6d6fe1c' *)
{attribute 'TcIecLibraryType'}
TYPE ST_xf09845edab6c83520d8d57def6d6fe1c : 
	STRUCT
		(* Generated from item 'clockTick0' *)
		nclockTick0 : UDINT;
		(* Generated from item 'clockTickH0' *)
		nclockTickH0 : UDINT;
		(* Generated from item 'stepSize0' *)
		fstepSize0 : LREAL;
		(* Generated from item 'clockTick1' *)
		nclockTick1 : UDINT;
		(* Generated from item 'clockTickH1' *)
		nclockTickH1 : UDINT;
		(* Generated from item 'tStart' *)
		ftStart : LREAL;
		(* Generated from item 'simTimeStep' *)
		esimTimeStep : E_SimTimeStep;
		(* Generated from item 'stopRequestedFlag' *)
		bstopRequestedFlag : BOOL;
		 {attribute 'hide'}
		_reserved1 : ARRAY [1..3] OF USINT;
		t : POINTER TO LREAL;
		(* Generated from item 'tArray' *)
		atArray : T_matrix2xdouble;
	END_STRUCT
END_TYPE

// DUTs/ST_RT_MODEL_vertical_levitation_control_T
(* Generated from type 'RT_MODEL_vertical_levitation_control_T' *)
{attribute 'TcIecLibraryType'}
{attribute 'pack_mode' := '1'}
TYPE ST_RT_MODEL_vertical_levitation_control_T : 
	STRUCT
		errorStatus : POINTER TO SINT;
		solverInfo : POINTER TO ST_ssSolverInfo;
		blockIO : POINTER TO ST_B_vertical_levitation_control_T;
		prevZCSigState : POINTER TO ST_PrevZCX_vertical_levitation_control_T;
		contStates : POINTER TO ST_X_vertical_levitation_control_T;
		periodicContStateIndices : POINTER TO DINT;
		periodicContStateRanges : POINTER TO LREAL;
		derivs : POINTER TO LREAL;
		inputs : POINTER TO ST_ExtU_vertical_levitation_control_T;
		outputs : POINTER TO ST_ExtY_vertical_levitation_control_T;
		contStateDisabled : POINTER TO ST_XDis_vertical_levitation_control_T;
		(* Generated from item 'zCCacheNeedsReset' *)
		bzCCacheNeedsReset : BOOL;
		(* Generated from item 'derivCacheNeedsReset' *)
		bderivCacheNeedsReset : BOOL;
		(* Generated from item 'CTOutputIncnstWithState' *)
		bCTOutputIncnstWithState : BOOL;
		 {attribute 'hide'}
		_reserved1 : UINT_8_40;
		(* Generated from item 'odeY' *)
		aodeY : T_matrix22xdouble;
		(* Generated from item 'odeF' *)
		aodeF : T_matrix22x4xdouble;
		(* Generated from item 'intgData' *)
		stintgData : ST_ODE4_IntgData;
		dwork : POINTER TO ST_DW_vertical_levitation_control_T;
		(* Generated from item 'Sizes' *)
		stSizes : ST_x08a7a7bbd0e5d629f7d70ceec84eacfe;
		 {attribute 'hide'}
		_reserved2 : UDINT;
		(* Generated from item 'Timing' *)
		stTiming : ST_xf09845edab6c83520d8d57def6d6fe1c;
	END_STRUCT
END_TYPE

// DUTs/T_matrix53xdouble
(* Generated from type 'matrix53xdouble' *)
{attribute 'TcIecLibraryType'}
TYPE T_matrix53xdouble : ARRAY [0..52] OF LREAL;
END_TYPE

// DUTs/T_matrix1007xdouble
(* Generated from type 'matrix1007xdouble' *)
{attribute 'TcIecLibraryType'}
TYPE T_matrix1007xdouble : ARRAY [0..1006] OF LREAL;
END_TYPE

// DUTs/T_matrix19xdouble
(* Generated from type 'matrix19xdouble' *)
{attribute 'TcIecLibraryType'}
TYPE T_matrix19xdouble : ARRAY [0..18] OF LREAL;
END_TYPE

// DUTs/T_matrix380xdouble
(* Generated from type 'matrix380xdouble' *)
{attribute 'TcIecLibraryType'}
TYPE T_matrix380xdouble : ARRAY [0..379] OF LREAL;
END_TYPE

// DUTs/T_matrix3xlogical
(* Generated from type 'matrix3xlogical' *)
{attribute 'TcIecLibraryType'}
{attribute 'BaseTypeGUID' := '18071995-0000-0000-0000-000000000030'}
TYPE T_matrix3xlogical : ARRAY [0..2] OF BOOL;
END_TYPE

// DUTs/ST_P_vertical_levitation_control_T
(* Generated from type 'P_vertical_levitation_control_T' *)
{attribute 'TcIecLibraryType'}
TYPE ST_P_vertical_levitation_control_T : 
	STRUCT
		(* Generated from item 'Airgaps_HEMS_DH10' *)
		aAirgaps_HEMS_DH10 : T_matrix53xdouble;
		(* Generated from item 'Current_to_force_coefficients_HEMS_DH10' *)
		aCurrent_to_force_coefficients_HEMS_DH10 : T_matrix1007xdouble;
		(* Generated from item 'Currents_HEMS_DH10' *)
		aCurrents_HEMS_DH10 : T_matrix19xdouble;
		(* Generated from item 'Force_to_current_coefficients_HEMS_DH10' *)
		aForce_to_current_coefficients_HEMS_DH10 : T_matrix380xdouble;
		(* Generated from item 'K_D_pit' *)
		fK_D_pit : LREAL;
		(* Generated from item 'K_D_roll' *)
		fK_D_roll : LREAL;
		(* Generated from item 'K_D_tot' *)
		fK_D_tot : LREAL;
		(* Generated from item 'K_F_init_pit' *)
		fK_F_init_pit : LREAL;
		(* Generated from item 'K_F_init_roll' *)
		fK_F_init_roll : LREAL;
		(* Generated from item 'K_F_init_tot' *)
		fK_F_init_tot : LREAL;
		(* Generated from item 'K_F_pit' *)
		fK_F_pit : LREAL;
		(* Generated from item 'K_F_roll' *)
		fK_F_roll : LREAL;
		(* Generated from item 'K_F_tot' *)
		fK_F_tot : LREAL;
		(* Generated from item 'K_I_init_pit' *)
		fK_I_init_pit : LREAL;
		(* Generated from item 'K_I_init_roll' *)
		fK_I_init_roll : LREAL;
		(* Generated from item 'K_I_init_tot' *)
		fK_I_init_tot : LREAL;
		(* Generated from item 'K_I_pit' *)
		fK_I_pit : LREAL;
		(* Generated from item 'K_I_roll' *)
		fK_I_roll : LREAL;
		(* Generated from item 'K_I_tot' *)
		fK_I_tot : LREAL;
		(* Generated from item 'K_P_pit' *)
		fK_P_pit : LREAL;
		(* Generated from item 'K_P_roll' *)
		fK_P_roll : LREAL;
		(* Generated from item 'K_P_tot' *)
		fK_P_tot : LREAL;
		(* Generated from item 'd_HEMS_to_HEMS' *)
		fd_HEMS_to_HEMS : LREAL;
		(* Generated from item 'enable_extra_roll_notch' *)
		fenable_extra_roll_notch : LREAL;
		(* Generated from item 'f_extra_roll_filter' *)
		ff_extra_roll_filter : LREAL;
		(* Generated from item 'g' *)
		fg : LREAL;
		(* Generated from item 'lift_off_time' *)
		flift_off_time : LREAL;
		(* Generated from item 'm' *)
		fm : LREAL;
		(* Generated from item 'notch_damp' *)
		fnotch_damp : LREAL;
		(* Generated from item 'notch_gmin' *)
		fnotch_gmin : LREAL;
		(* Generated from item 'pitch_target' *)
		fpitch_target : LREAL;
		(* Generated from item 'r_motor_left_com' *)
		ar_motor_left_com : T_matrix3xdouble;
		(* Generated from item 'r_motor_right_com' *)
		ar_motor_right_com : T_matrix3xdouble;
		(* Generated from item 'r_pitch_hems' *)
		ar_pitch_hems : T_matrix4xdouble;
		(* Generated from item 'r_roll_hems' *)
		ar_roll_hems : T_matrix4xdouble;
		(* Generated from item 'roll_target' *)
		froll_target : LREAL;
		(* Generated from item 'z_initial_lift_off' *)
		fz_initial_lift_off : LREAL;
		(* Generated from item 'z_manual_target' *)
		fz_manual_target : LREAL;
		(* Generated from item 'z_mismatch_D' *)
		fz_mismatch_D : LREAL;
		(* Generated from item 'z_mismatch_F' *)
		fz_mismatch_F : LREAL;
		(* Generated from item 'z_mismatch_I' *)
		fz_mismatch_I : LREAL;
		(* Generated from item 'z_mismatch_P' *)
		fz_mismatch_P : LREAL;
		(* Generated from item 'feed_forward_ems_ON' *)
		bfeed_forward_ems_ON : BOOL;
		(* Generated from item 'feed_fwd_motor_roll_ON' *)
		bfeed_fwd_motor_roll_ON : BOOL;
		(* Generated from item 'levi_operational' *)
		blevi_operational : BOOL;
		(* Generated from item 'lift_off_enabled' *)
		blift_off_enabled : BOOL;
		(* Generated from item 'mismatch_enabled' *)
		bmismatch_enabled : BOOL;
		(* Generated from item 'mismatch_specific_enabler' *)
		amismatch_specific_enabler : T_matrix3xlogical;
		(* Generated from item 'pitch_ON' *)
		bpitch_ON : BOOL;
		(* Generated from item 'roll_ON' *)
		broll_ON : BOOL;
		(* Generated from item 'roll_filter_enabled' *)
		broll_filter_enabled : BOOL;
		(* Generated from item 'total_ON' *)
		btotal_ON : BOOL;
		 {attribute 'hide'}
		_reserved1 : UDINT;
		(* Generated from item 'DiscreteDerivative_ICPrevScaledInput' *)
		fDiscreteDerivative_ICPrevScaledInput : LREAL;
		(* Generated from item 'PIDController_InitialConditionForFilter' *)
		fPIDController_InitialConditionForFilter : LREAL;
		(* Generated from item 'PIDController_InitialConditionForFilter_a' *)
		fPIDController_InitialConditionForFilter_a : LREAL;
		(* Generated from item 'PIDController_InitialConditionForFilter_j' *)
		fPIDController_InitialConditionForFilter_j : LREAL;
		(* Generated from item 'PIDController_InitialConditionForIntegrator' *)
		fPIDController_InitialConditionForIntegrator : LREAL;
		(* Generated from item 'PIDController_InitialConditionForIntegrator_m' *)
		fPIDController_InitialConditionForIntegrator_m : LREAL;
		(* Generated from item 'PIDController_InitialConditionForIntegrator_p' *)
		fPIDController_InitialConditionForIntegrator_p : LREAL;
		(* Generated from item 'PIDController_LowerSaturationLimit' *)
		fPIDController_LowerSaturationLimit : LREAL;
		(* Generated from item 'PIDController_LowerSaturationLimit_n' *)
		fPIDController_LowerSaturationLimit_n : LREAL;
		(* Generated from item 'PIDController_LowerSaturationLimit_e' *)
		fPIDController_LowerSaturationLimit_e : LREAL;
		(* Generated from item 'PIDController_UpperSaturationLimit' *)
		fPIDController_UpperSaturationLimit : LREAL;
		(* Generated from item 'PIDController_UpperSaturationLimit_n' *)
		fPIDController_UpperSaturationLimit_n : LREAL;
		(* Generated from item 'PIDController_UpperSaturationLimit_g' *)
		fPIDController_UpperSaturationLimit_g : LREAL;
		(* Generated from item 'Constant1_Value' *)
		fConstant1_Value : LREAL;
		(* Generated from item 'Constant1_Value_b' *)
		fConstant1_Value_b : LREAL;
		(* Generated from item 'Constant1_Value_e' *)
		fConstant1_Value_e : LREAL;
		(* Generated from item 'Constant4_Value' *)
		fConstant4_Value : LREAL;
		(* Generated from item 'Constant4_Value_e' *)
		fConstant4_Value_e : LREAL;
		(* Generated from item 'UnitDelay_InitialCondition' *)
		fUnitDelay_InitialCondition : LREAL;
		(* Generated from item 'Integrator1_IC' *)
		fIntegrator1_IC : LREAL;
		(* Generated from item 'Constant5_Value' *)
		fConstant5_Value : LREAL;
		(* Generated from item 'Switch1_Threshold' *)
		fSwitch1_Threshold : LREAL;
		(* Generated from item 'Constant7_Value' *)
		fConstant7_Value : LREAL;
		(* Generated from item 'Switch1_Threshold_i' *)
		fSwitch1_Threshold_i : LREAL;
		(* Generated from item 'sat_enabled_Value' *)
		fsat_enabled_Value : LREAL;
		(* Generated from item 'Constant8_Value' *)
		fConstant8_Value : LREAL;
		(* Generated from item 'Constant9_Value' *)
		fConstant9_Value : LREAL;
		(* Generated from item 'Switch2_Threshold' *)
		fSwitch2_Threshold : LREAL;
		(* Generated from item 'Delay_InitialCondition' *)
		fDelay_InitialCondition : LREAL;
		(* Generated from item 'UnitDelay1_InitialCondition' *)
		fUnitDelay1_InitialCondition : LREAL;
		(* Generated from item 'Constant_Value' *)
		fConstant_Value : LREAL;
		(* Generated from item 'stop_div_by_zero_Threshold' *)
		fstop_div_by_zero_Threshold : LREAL;
		(* Generated from item 'error_integrator_IC' *)
		ferror_integrator_IC : LREAL;
		(* Generated from item 'time_integrator_IC' *)
		ftime_integrator_IC : LREAL;
		(* Generated from item 'Constant_Value_c' *)
		fConstant_Value_c : LREAL;
		(* Generated from item 'tau_Gain' *)
		ftau_Gain : LREAL;
		(* Generated from item 'Bias_Bias' *)
		fBias_Bias : LREAL;
		(* Generated from item 'two_Gain' *)
		ftwo_Gain : LREAL;
		(* Generated from item 'one_Gain' *)
		fone_Gain : LREAL;
		(* Generated from item 'UnitDelay1_InitialCondition_m' *)
		fUnitDelay1_InitialCondition_m : LREAL;
		(* Generated from item 'TSamp_WtEt' *)
		fTSamp_WtEt : LREAL;
		(* Generated from item 'Gain_Gain' *)
		fGain_Gain : LREAL;
		(* Generated from item 'f_roll_n_Value' *)
		ff_roll_n_Value : LREAL;
		(* Generated from item 'tau_Gain_h' *)
		ftau_Gain_h : LREAL;
		(* Generated from item 'Bias_Bias_j' *)
		fBias_Bias_j : LREAL;
		(* Generated from item 'damp_roll_notch_Value' *)
		fdamp_roll_notch_Value : LREAL;
		(* Generated from item 'two_Gain_h' *)
		ftwo_Gain_h : LREAL;
		(* Generated from item 'g_roll_notch_Value' *)
		fg_roll_notch_Value : LREAL;
		(* Generated from item 'one_Gain_l' *)
		fone_Gain_l : LREAL;
		(* Generated from item 'UnitDelay1_InitialCondition_h' *)
		fUnitDelay1_InitialCondition_h : LREAL;
		(* Generated from item 'tau_Gain_b' *)
		ftau_Gain_b : LREAL;
		(* Generated from item 'Bias_Bias_c' *)
		fBias_Bias_c : LREAL;
		(* Generated from item 'two_Gain_f' *)
		ftwo_Gain_f : LREAL;
		(* Generated from item 'one_Gain_g' *)
		fone_Gain_g : LREAL;
		(* Generated from item 'UnitDelay1_InitialCondition_c' *)
		fUnitDelay1_InitialCondition_c : LREAL;
		(* Generated from item 'Switch_Threshold' *)
		fSwitch_Threshold : LREAL;
		(* Generated from item 'Gain1_Gain' *)
		fGain1_Gain : LREAL;
		(* Generated from item 'tau_Gain_d' *)
		ftau_Gain_d : LREAL;
		(* Generated from item 'Bias_Bias_g' *)
		fBias_Bias_g : LREAL;
		(* Generated from item 'two_Gain_fc' *)
		ftwo_Gain_fc : LREAL;
		(* Generated from item 'one_Gain_f' *)
		fone_Gain_f : LREAL;
		(* Generated from item 'UnitDelay1_InitialCondition_ci' *)
		fUnitDelay1_InitialCondition_ci : LREAL;
		(* Generated from item 'dist_enabled_Value' *)
		fdist_enabled_Value : LREAL;
		(* Generated from item 'UnitDelay1_InitialCondition_n' *)
		fUnitDelay1_InitialCondition_n : LREAL;
		(* Generated from item 'Constant_Value_e' *)
		fConstant_Value_e : LREAL;
		(* Generated from item 'stop_div_by_zero_Threshold_g' *)
		fstop_div_by_zero_Threshold_g : LREAL;
		(* Generated from item 'UnitDelay1_InitialCondition_nc' *)
		fUnitDelay1_InitialCondition_nc : LREAL;
		(* Generated from item 'Constant_Value_a' *)
		fConstant_Value_a : LREAL;
		(* Generated from item 'stop_div_by_zero_Threshold_p' *)
		fstop_div_by_zero_Threshold_p : LREAL;
		(* Generated from item 'ZeroGain_Gain' *)
		fZeroGain_Gain : LREAL;
		(* Generated from item 'ZeroGain_Gain_m' *)
		fZeroGain_Gain_m : LREAL;
		(* Generated from item 'ZeroGain_Gain_a' *)
		fZeroGain_Gain_a : LREAL;
		(* Generated from item 'Constant_Value_o' *)
		fConstant_Value_o : LREAL;
		(* Generated from item 'Bias1_Bias' *)
		fBias1_Bias : LREAL;
		(* Generated from item 'Gain_Gain_p' *)
		fGain_Gain_p : LREAL;
		(* Generated from item 'UnitDelay2_InitialCondition' *)
		fUnitDelay2_InitialCondition : LREAL;
		(* Generated from item 'Bias1_Bias_d' *)
		fBias1_Bias_d : LREAL;
		(* Generated from item 'Gain_Gain_c' *)
		fGain_Gain_c : LREAL;
		(* Generated from item 'UnitDelay2_InitialCondition_j' *)
		fUnitDelay2_InitialCondition_j : LREAL;
		(* Generated from item 'Bias1_Bias_l' *)
		fBias1_Bias_l : LREAL;
		(* Generated from item 'Gain_Gain_d' *)
		fGain_Gain_d : LREAL;
		(* Generated from item 'UnitDelay2_InitialCondition_p' *)
		fUnitDelay2_InitialCondition_p : LREAL;
		(* Generated from item 'Bias1_Bias_j' *)
		fBias1_Bias_j : LREAL;
		(* Generated from item 'Gain_Gain_a' *)
		fGain_Gain_a : LREAL;
		(* Generated from item 'UnitDelay2_InitialCondition_a' *)
		fUnitDelay2_InitialCondition_a : LREAL;
		(* Generated from item 'Constant10_Value' *)
		fConstant10_Value : LREAL;
		(* Generated from item 'Constant6_Value' *)
		fConstant6_Value : LREAL;
		(* Generated from item 'Constant7_Value_o' *)
		fConstant7_Value_o : LREAL;
		(* Generated from item 'Constant8_Value_h' *)
		fConstant8_Value_h : LREAL;
		(* Generated from item 'Constant9_Value_p' *)
		fConstant9_Value_p : LREAL;
		(* Generated from item 'Integrator2_IC' *)
		fIntegrator2_IC : LREAL;
		(* Generated from item 'IsPeak1_Threshold' *)
		fIsPeak1_Threshold : LREAL;
		(* Generated from item 'Switch2_Threshold_n' *)
		fSwitch2_Threshold_n : LREAL;
		(* Generated from item 'Constant2_Value' *)
		fConstant2_Value : LREAL;
		(* Generated from item 'Constant2_Value_e' *)
		fConstant2_Value_e : LREAL;
		(* Generated from item 'Constant2_Value_d' *)
		fConstant2_Value_d : LREAL;
		(* Generated from item 'Delay1_InitialCondition' *)
		fDelay1_InitialCondition : REAL;
		(* Generated from item 'wasfmenabledlastrun_Threshold' *)
		fwasfmenabledlastrun_Threshold : REAL;
		(* Generated from item 'hard_disable_fmm_Gain' *)
		fhard_disable_fmm_Gain : REAL;
		(* Generated from item 'usefmornot_Threshold' *)
		fusefmornot_Threshold : REAL;
		(* Generated from item 'Memory_InitialCondition' *)
		bMemory_InitialCondition : BOOL;
		(* Generated from item 'Memory_InitialCondition_m' *)
		bMemory_InitialCondition_m : BOOL;
		(* Generated from item 'Memory_InitialCondition_n' *)
		bMemory_InitialCondition_n : BOOL;
		(* Generated from item 'Switch_Threshold_c' *)
		nSwitch_Threshold_c : USINT;
		 {attribute 'hide'}
		_reserved2 : UDINT;
	END_STRUCT
END_TYPE

// DUTs/E_ModuleCaller
(* Generated from type 'TcMgSdk.ModuleCaller' *)
{attribute 'TcIecLibraryType'}
TYPE E_ModuleCaller : (
	CyclicTask:=0, 	(* Add to the specified cyclic caller tasks. *)
	Module:=1	(* Don't add to cyclic callers. The module can be called from other TwinCAT modules (e. g. a PLC). *)
) DINT;
END_TYPE

// DUTs/E_CallerVerification
(* Generated from type 'TcMgSdk.CallerVerification' *)
{attribute 'TcIecLibraryType'}
TYPE E_CallerVerification : (
	Default:=0, 	(* Verify the caller task only if the "ModuleCaller" parameter is set to "Module" but not when added to cyclic caller tasks. *)
	Always:=1, 	(* Always verify the caller context to prevent concurrent execution of model code and corresponding DataArea mappings. *)
	Never:=2	(* Skip caller verification to reduce execution times. *)
) DINT;
END_TYPE

// DUTs/E_StepSizeAdaptation
(* Generated from type 'TcMgSdk.StepSizeAdaptation' *)
{attribute 'TcIecLibraryType'}
TYPE E_StepSizeAdaptation : (
	RequireMatchingTaskCycleTime:=0, 	(* Don't accept task cycle times other than the Simulink step sizes. *)
	UseTaskCycleTime:=1, 	(* Adapt the Smulink step sizes to the task cycle times. *)
	UseModelStepSize:=2	(* Keep the Smulink step sizes, independent of the callers cycle time. *)
) DINT;
END_TYPE

// DUTs/E_ExecutionSequence1
(* Generated from type 'TcMgSdk.ExecutionSequence1' *)
{attribute 'TcIecLibraryType'}
TYPE E_ExecutionSequence1 : (
	UpdateBeforeOutputMapping:=0, 	(* Input mapping -> State and output update -> Output mapping -> ADS processing *)
	IoAtTaskBegin:=1	(* Input mapping -> Code execution -> Output update -> ADS processing *)
) DINT;
END_TYPE

// DUTs/E_FpExcptCtrlSet
(* Generated from type 'TcMgSdk.FpExcptCtrlSet' *)
{attribute 'TcIecLibraryType'}
TYPE E_FpExcptCtrlSet : (
	CallerExceptions:=1, 	(* Use the floating point exception settings provided by the caller *)
	ThrowExceptions:=3, 	(* Enable floating point exceptions on invalid operations and divisions by zero *)
	SuppressExceptions:=5	(* Disable floating point exceptions. *)
) USINT;
END_TYPE

// DUTs/ST_TcMatSim_ModuleGeneratorInfo
(* Generated from type 'TcMatSim.ModuleGeneratorInfo' *)
{attribute 'TcIecLibraryType'}
TYPE ST_TcMatSim_ModuleGeneratorInfo : 
	STRUCT
		(* Generated from item 'MatlabVersion' *)
		nMatlabVersion : ARRAY [0..3] OF UDINT;
		(* Generated from item 'TE140xVersion' *)
		nTE140xVersion : ARRAY [0..3] OF UDINT;
	END_STRUCT
END_TYPE

// DUTs/ST_TcMatSim_SimulinkModelInfo
(* Generated from type 'TcMatSim.SimulinkModelInfo' *)
{attribute 'TcIecLibraryType'}
TYPE ST_TcMatSim_SimulinkModelInfo : 
	STRUCT
		(* Generated from item 'ModelName' *)
		{attribute 'GUID' := '18071995-0000-0000-0000-00010000007F'}
		sModelName : STRING(127);
		(* Generated from item 'SimulinkVersion' *)
		nSimulinkVersion : ARRAY [0..3] OF UDINT;
		(* Generated from item 'ModelVersion' *)
		nModelVersion : ARRAY [0..3] OF UDINT;
		(* Generated from item 'ModelChecksum' *)
		nModelChecksum : ARRAY [0..3] OF UDINT;
	END_STRUCT
END_TYPE

// DUTs/E_ParameterSharingType
(* Generated from type 'ParameterSharingType' *)
{attribute 'TcIecLibraryType'}
TYPE E_ParameterSharingType : (
	Define:=0, 	(* This module instance defines the parameter values for all further instances of this module class. Exactly one instance of this module class must use this option. *)
	Inherit:=1	(* This module instance inherits the parameter values from the instance of this module class configured to "Define" the parameter values. Model parameters configured at this instsance are ignored. *)
) DINT;
END_TYPE

// DUTs/ST_FB_vertical_levitation_control_TcCOM_InitStruct
{attribute 'TcIecLibraryType'}
TYPE ST_FB_vertical_levitation_control_TcCOM_InitStruct : 
	STRUCT
		{attribute 'GUID' := '18071995-0000-0000-0000-000000000061'}
		eObjState : TCOM_STATE := TCOM_STATE.TCOM_STATE_OP;
		{attribute 'GUID' := '18071995-0000-0000-0000-00010000007F'}
		sObjName : STRING(127);
		{attribute 'GUID' := '18071995-0000-0000-0000-00000000000F'}
		nOid : OTCID := 4294967295;
		{attribute 'GUID' := '18071995-0000-0000-0000-00000000000F'}
		nTaskOid : OTCID;
		nTaskSortOrder : UDINT;
		{attribute 'GUID' := '8007AE3B-86BB-40F2-B385-EF87FCC239A4'}
		eTraceLevelMax : TcTraceLevel := TcTraceLevel.tlInfo;
		eModuleCaller : E_ModuleCaller := E_ModuleCaller.CyclicTask;
		eCallerVerification : E_CallerVerification := E_CallerVerification.Default;
		eStepSizeAdaptation : E_StepSizeAdaptation := E_StepSizeAdaptation.RequireMatchingTaskCycleTime;
		eExecutionSequence : E_ExecutionSequence1 := E_ExecutionSequence1.UpdateBeforeOutputMapping;
		bExecute : BOOL := TRUE;
		 {attribute 'hide'}
		_reserved1 : ARRAY [1..3] OF USINT;
		{attribute 'GUID' := '18071995-0000-0000-0000-000000000061'}
		eAccessLockState : TCOM_STATE := TCOM_STATE.TCOM_STATE_OP;
		eInitExceptionHandling : E_FpExcptCtrlSet := E_FpExcptCtrlSet.CallerExceptions;
		eUpdateExceptionHandling : E_FpExcptCtrlSetEx := E_FpExcptCtrlSetEx.CallerExceptions;
		 {attribute 'hide'}
		_reserved2 : UINT;
		stModuleGeneratorInfo : ST_TcMatSim_ModuleGeneratorInfo;
		stSimulinkModelInfo : ST_TcMatSim_SimulinkModelInfo;
		evertical_levitation_control_P_Sharing : E_ParameterSharingType := E_ParameterSharingType.Define;
		 {attribute 'hide'}
		_reserved3 : UDINT;
		stvertical_levitation_control_P : ST_P_vertical_levitation_control_T := (aAirgaps_HEMS_DH10 := [4.0,4.5,5.0,5.5,6.0,6.5,7.0,7.5,8.0,8.5,9.0,9.5,10.0,10.5,11.0,11.5,12.0,12.5,13.0,13.5,14.0,14.5,15.0,15.5,16.0,16.5,17.0,17.5,18.0,18.5,19.0,19.5,20.0,20.5,21.0,21.5,22.0,22.5,23.0,23.5,24.0,24.5,25.0,25.5,26.0,26.5,27.0,27.5,28.0,28.5,29.0,29.5,30.0], aCurrent_to_force_coefficients_HEMS_DH10 := [-0.760550596997102,-837774978.924559,1103552349.97731,4926.68060549225,600.745180207589,26.4958253766194,-0.349817285754332,-2.33531126074652,-0.746391275559456,0.0452051379913167,0.0475267467399872,0.000763448701129376,-0.00148612074185778,-4.1373783940125e-05,2.54091130676406e-05,5.58202265723376e-07,-2.25069518403088e-07,-2.51299121293643e-09,8.03655499171807e-10,0.00222886398979671,-781584939.428744,1185623768.70936,4724.96313801348,576.330957904419,25.5365281690957,1.04382709119927,-2.00500220404158,-0.827664241880529,0.0269583906734128,0.0502714801965582,0.0012398294770021,-0.00153778840410471,-4.79454542738909e-05,2.58988547307712e-05,6.04621600825917e-07,-2.26729512593462e-07,-2.64603751283049e-09,8.01941299546001e-10,8.20967090784988,-793775204.854193,988504041.693301,4484.99323395838,546.332827164944,34.262779909026,5.33983916658022,-3.43181093093475,-1.21527130693203,0.140205631115838,0.0669598543719415,-0.00319377154108582,-0.00191255775299226,4.16449390925401e-05,3.03202718251557e-05,-2.89773590239561e-07,-2.51780680865415e-07,8.33751060554298e-10,8.5164543979002e-10,4.91155870653422,-688851949.530325,1061093336.6486,4276.5127590897,526.685025821111,31.0414021633379,2.92874595808965,-2.56302578568842,-0.78296775983484,0.0687552895017945,0.038292766760148,-0.000368422276595244,-0.00094970815768204,-1.58168336829756e-05,1.29809285858825e-05,2.86507185707269e-07,-9.28681345703773e-08,-1.41538546142088e-09,2.71614553604299e-10,2594.94736126,56387057.9896639,1335190054.27943,6.29326885131012,501.666842127006,26.4255811830483,3.65493500297621,-2.09906087653859,-0.805400418343247,0.0581197556296744,0.0384786469310301,-0.000538772597150557,-0.000937679490128882,-5.41801539699554e-06,1.25621285062245e-05,1.39793360429851e-07,-8.766972076382e-08,-7.36849406917905e-10,2.48730979937201e-10,-11.1997313775952,536863109.612347,-1048023701.17251,3870.28344745263,482.819122993976,32.6421713982239,6.23096751415027,-2.72367040873607,-1.14907544965355,0.097747240435102,0.0611501676941498,-0.00196552840212844,-0.00173191095353189,2.26913988629049e-05,2.75570213383152e-05,-1.4007877716167e-07,-2.30966016665903e-07,3.57837307374209e-10,7.90051947799413e-10,-7.51793938344168,661079007.553125,-904353413.279481,3702.80657812258,462.814449420192,27.9905871721004,5.58812419786516,-2.00844015298035,-0.987450458014825,0.0521213877010948,0.0496606189400889,-0.000379447753263228,-0.00132354005877068,-7.68799022036313e-06,1.98025731510788e-05,1.5690501799561e-07,-1.56495519101817e-07,-7.90495881424282e-10,5.07373296269548e-10,-7.22955387977831,621575764.988751,-883006736.900246,3541.82411212497,434.046747994495,24.531742402371,9.48675197130834,-1.45583692472823,-1.45088074708644,0.0200080267075973,0.0781580247600355,0.000550599698380177,-0.00227216464142579,-2.17914285916637e-05,3.7052387613234e-05,2.63339401078147e-07,-3.16913933374467e-07,-1.10424215456079e-09,1.10161317980292e-09,-9.96865774337514,607884998.305149,-845512487.935064,3385.62203158026,422.168274217811,25.8960675386644,8.51054858166488,-1.64099191225096,-1.30882114678658,0.0374204060750377,0.0703441237800478,-0.000166351044879653,-0.00204877214840399,-7.51692528047424e-06,3.35123180203377e-05,1.27138788623499e-07,-2.87383522437384e-07,-6.04115946556581e-10,1.0006343077375e-09,-8.81956277273346,595537984.996708,-810114571.570841,3240.89254695914,407.872890364362,21.5398973608528,6.6764027168254,-0.774427230214992,-0.99226846484053,-0.0268268422051902,0.0492618685257872,0.00218724873997593,-0.00133379647308237,-5.24866413560896e-05,2.05317683016023e-05,5.55337604637202e-07,-1.67748475289645e-07,-2.20480124404583e-09,5.62418315193606e-10,0.694918644261154,-576974338.80199,825580840.504478,3122.47714800563,392.281669122699,10.019558146974,4.30002400507528,0.847353938967864,-0.587480300609353,-0.129355497888877,0.0218076610817335,0.00564539022075976,-0.000377424149812828,-0.000116148705639108,2.67875471240442e-06,1.15453712882485e-06,1.05267686174407e-09,-4.44907198786716e-09,-6.97410305926543e-11,0.313563918721904,-559646477.538789,807368355.00881,2987.20306175122,377.518380911724,8.53067008504387,3.80020234918953,1.08440658110241,-0.4907231203257,-0.139141627285258,0.0163634631818611,0.00575398924487597,-0.000233233123015646,-0.00011424874822487,7.58594140881123e-07,1.10536022955494e-06,1.31115118955816e-08,-4.17029055984419e-09,-9.65145890961053e-11,-1.03163877693509,544564533.701197,-785452367.025036,2855.64057150643,364.939117626786,9.51379776696453,3.15774859738957,0.911744893797488,-0.379574362931593,-0.124670313163687,0.00926343888267286,0.00521192533074427,2.73988380283842e-06,-0.000104040982030531,-3.50094773407731e-06,1.0105075173277e-06,5.24234914012352e-08,-3.82435802683389e-09,-2.41136809595459e-10,12.6676979041015,535989148.015584,-790032874.129763,2757.99960423547,355.944387701876,5.27244916540905,-1.21327195252169,1.04748993520978,0.18876327356635,-0.113915690861857,-0.0238491255040581,0.00442774959187147,0.00103716107982964,-8.46371695325393e-05,-2.12948789287141e-05,7.97711509816267e-07,2.10498933822655e-07,-2.95320694063708e-09,-8.05422194198633e-10,7.91955951469276,519601123.644615,-756401770.66565,2636.14908640798,350.523943402419,8.56423013740456,-2.16558762861436,0.478831438179988,0.250536276102788,-0.0714878470439507,-0.0248323687225368,0.00287912156176228,0.00100773873075833,-5.51931118404583e-05,-2.00378985108881e-05,5.18122676685497e-07,1.94525177360337e-07,-1.9084823974239e-09,-7.36013342601176e-10,3.98692554903957,498903809.137368,-726986300.636497,2519.00775985004,337.671905876894,8.85921810727892,-1.67174343632598,0.606917700911879,0.214658065453568,-0.0843666029406792,-0.0229290811855915,0.0034101512610016,0.000946518182117042,-6.59995473925995e-05,-1.89320840630632e-05,6.25138379685104e-07,1.84273363897491e-07,-2.31945258984255e-09,-6.98207396938304e-10,1.64121632675127,590799317.305316,-642824599.798975,2416.23994445287,326.677023630802,10.3135751393108,-1.69924438026672,0.322144310419216,0.267621925223191,-0.0597548384154244,-0.0280014309008958,0.00241947609489079,0.00115478238984662,-4.58931700174555e-05,-2.31851625416197e-05,4.25502306819769e-07,2.26630389661337e-07,-1.54980091170952e-09,-8.6185078249918e-10,0.711231119216587,-1207893473.69676,786746134.208984,2314.63424329605,315.83455160256,11.5652163748054,-1.19346386674732,-0.00163515664404085,0.174202829300681,-0.0301369141234384,-0.0202458952621126,0.00121113051767515,0.000848306477965107,-2.12511913172145e-05,-1.70164439689121e-05,1.80121999849654e-07,1.65590904522222e-07,-6.01491838530031e-10,-6.26777452657362e-10,-4.93055620435076,-487503965.429625,655672101.603393,2229.25152065123,303.226752892414,7.62237819649985,-2.06860456516372,0.528110245813339,0.300648742155722,-0.0643316297518648,-0.0270999208436176,0.00242769185331215,0.00104746351604381,-4.48755270651864e-05,-2.02776678855788e-05,4.12264393659654e-07,1.93770352327407e-07,-1.49944521421776e-09,-7.26091424325227e-10,-2.96600021577164,-577446118.343753,595498737.165061,2137.41689585903,294.097311059148,6.12531599110267,-2.50197423855597,0.864126284643337,0.39191538836475,-0.0879565643979353,-0.0339191933247201,0.00320645273695014,0.00129745522697844,-5.79702832912213e-05,-2.50425850924291e-05,5.20992360202213e-07,2.38970891693309e-07,-1.8530639217935e-09,-8.94378189868182e-10,-9.11310783779881,-393466671.273951,1368025494.94802,2058.76941972191,280.718886587965,11.086002598274,0.78404162683319,-0.043311213338657,-0.169607415510759,-0.0290814512510207,0.00502058583376664,0.00133714371004766,-5.51428509683742e-05,-2.65601159653698e-05,-1.44676401847714e-07,2.52935987588952e-07,7.56733748799219e-09,-9.38627430747115e-10,-4.2149241728059e-11,-4.02478369374427,-419552228.416979,666398856.165128,1970.05722874854,273.12314656252,6.45323922466905,-2.61006619645486,0.699810046737068,0.436755597593477,-0.0701248667194684,-0.036466238056829,0.00242995444054236,0.00136544432403539,-4.15412728984944e-05,-2.59799597856772e-05,3.53359364565495e-07,2.45330283060203e-07,-1.19399038333151e-09,-9.10893528169556e-10,-2.78985180044047,-421749515.963403,627150546.782587,1892.82716832413,264.597914927991,5.71325736387936,-2.9504938308236,0.79564678817595,0.502975013512827,-0.0770056154890885,-0.041176034361541,0.00273432641369968,0.00153901763092019,-4.87066517567256e-05,-2.94085434268775e-05,4.34583371741474e-07,2.79417907265817e-07,-1.54209093851923e-09,-1.04401895160885e-09,-11.0749863372858,323024657.001645,-1442903911.45917,1795.13267411418,252.972212044683,11.1948605823352,0.0832921629743774,-0.477900146975261,-0.0792420038493669,0.0353342571034955,0.00545071899892178,-0.00178023707791573,-0.000261413587015873,4.24750570199075e-05,6.30940688172939e-06,-4.67178489321753e-07,-7.08289691579036e-08,1.92562206718749e-09,2.97302194377254e-10,-4.11089115119773,-405736972.174835,599536636.462214,1751.77615628515,247.971430820694,5.53113017077834,-3.40194688568508,0.586564339128313,0.538462494858911,-0.0516052350340621,-0.0409899686016586,0.00159301637216167,0.00147046879788508,-2.42166555205679e-05,-2.73455484008934e-05,1.8272028239922e-07,2.54847438804131e-07,-5.46833323489066e-10,-9.38797245489454e-10,-5.094441725813,267347243.370697,-745422013.046013,1668.46136960569,235.405235063912,6.21470901547794,-0.62723858051798,0.880556808753658,0.223953565808477,-0.0861853468815011,-0.0238275984115981,0.0031186848104217,0.000961928251814803,-5.64418931970624e-05,-1.8966904680682e-05,5.09227890040404e-07,1.82862743154715e-07,-1.81955040781975e-09,-6.88162416638629e-10,3.93452621280867,386280535.707499,-611683998.56737,1619.83357996186,228.947276372313,4.89273035090957,-2.35222592604079,0.597992608381673,0.400922104255278,-0.0490117008791364,-0.0315310172839264,0.00144397025790875,0.00113327396312414,-2.08030651162903e-05,-2.09591214190029e-05,1.46560205410556e-07,1.93998714664476e-07,-4.01149974298634e-10,-7.10116712081297e-10,-4.42658521053589,-390536168.056176,637251581.011691,1560.77250252062,222.871200649395,3.40179042396259,-3.26301068923526,0.845645153621507,0.540181974333895,-0.0674649765450875,-0.0407659842334083,0.00216028774661521,0.00145725136145249,-3.54410756286128e-05,-2.71002347970254e-05,2.94857325086111e-07,2.52964037026926e-07,-9.85762213676321e-10,-9.3383122532233e-10,1.04270777521884,366286808.046656,-560859350.028844,1496.24882673917,213.815428028719,5.70723833517461,-1.48595989638926,0.470075796699391,0.278943853265913,-0.0402083603381079,-0.0232528706152899,0.00115281794369983,0.000846822909659337,-1.57107118169846e-05,-1.56853210161622e-05,1.01065272639095e-07,1.44885666107582e-07,-2.38030341447444e-10,-5.28715264745011e-10,3.68510819036719,-351761206.447311,858168256.600514,1433.54464713959,206.49101382676,5.38204401554629,-0.773809481741972,0.748098488440298,0.205555347424097,-0.0692765535235047,-0.0195442877092045,0.00243437433896036,0.000748082355092462,-4.33498512106815e-05,-1.42681565877783e-05,3.88070621505828e-07,1.34533580339005e-07,-1.38299731493592e-09,-4.98578027769054e-10,0.0754314723344674,-468571936.12136,-489243229.182402,1386.25537600482,200.099704607586,6.98489702131971,-0.544575659778846,0.191898679382798,0.104819467686376,-0.0203528005618932,-0.00997416583374995,0.000492659647694064,0.000356059112308431,-4.32588750331456e-06,-6.26952968131642e-06,2.1820820168629e-09,5.48208477821011e-08,1.04087018053142e-10,-1.90102777671726e-10,0.753954075978208,-1530292977.4048,-453997267.103364,1336.51138471102,196.165400427285,6.19266636661465,-1.12682525138909,0.376888331315186,0.190767311041754,-0.0369730888443862,-0.0160813790286187,0.0011890976052674,0.000583442596220964,-1.89697114196547e-05,-1.074915306239e-05,1.51943554187314e-07,9.88629596280787e-08,-4.87412660616997e-10,-3.59646981627663e-10,-0.297306919386193,-340120922.210493,628635768.138964,1287.57494076467,187.715268380531,6.50946927000666,-0.821666952888799,0.144245438462609,0.140917935706808,-0.0110839266346784,-0.0112952732132428,2.3758571027579e-05,0.000373494842859396,6.32124832783138e-06,-6.22540348683321e-06,-1.10848153872724e-07,5.19985344590937e-08,5.59281200360797e-10,-1.73293418258354e-10,1.0153933654993,-436465698.815783,-404331140.071419,1240.37827388261,181.231420429795,5.36981188404722,-0.256268795795976,0.440739700994461,0.0797857756645116,-0.0387040796005867,-0.008524424817447,0.00121293949457448,0.00031733361039804,-1.92585420497746e-05,-5.7876158911218e-06,1.55633287431514e-07,5.23775134978063e-08,-5.08884704501226e-10,-1.87748459245433e-10,-0.904613320386338,-418192057.60663,884428245.880484,1196.7800939288,174.400271635929,6.37450490115846,0.010046881989716,0.169159689682992,0.0277562208933746,-0.0164134638998619,-0.00418432856948087,0.000345799171480726,0.000144207756853181,-1.7597593695619e-06,-2.23433414003203e-06,-1.99801250650472e-08,1.63563065796601e-08,1.80298549536879e-10,-4.55770698015953e-11,0.704118195026607,-413524376.163251,-425977647.347842,1155.43210726019,169.703138391946,5.32231517325394,-0.0849078430893835,0.327569116707867,0.0501882678216723,-0.0278812691183175,-0.00593210969295418,0.00079655727578361,0.000213943488814453,-1.12879838925525e-05,-3.70805430191258e-06,8.04753677370831e-08,3.18376394768116e-08,-2.31152626557455e-10,-1.08747357933583e-10,0.749283703487053,-413931819.019776,881705064.82772,1111.17951449184,163.835350015503,6.0224611671284,-0.0767990539414558,0.243365060632776,0.0635466936886884,-0.0232536460652307,-0.00718919407579212,0.0006499164707373,0.000264303871251472,-8.47086438309326e-06,-4.69938620962002e-06,5.10729394774869e-08,4.12732820569231e-08,-1.07194589966151e-10,-1.43453762416732e-10,-0.448607370323945,-1064151748.47792,595066644.988328,1074.75383236036,158.392081932132,5.60894552363778,0.048548456917106,0.218559748109651,0.026342576999842,-0.0193398526902755,-0.00374903218624757,0.000493030813596321,0.00012621789118172,-5.64099225166682e-06,-1.94138038401012e-06,2.71531523990628e-08,1.43460641807665e-08,-3.04497313925198e-11,-4.11629327327894e-11,0.499487676901722,1105914887.44282,-533493396.835336,1038.24688237295,153.751814562601,5.25541896592344,-0.0644027183265858,0.218940245560314,0.042890143090272,-0.0169890782635692,-0.00470815319184722,0.000348397122366654,0.000156556179264017,-2.00635787774285e-06,-2.46981393835643e-06,-1.42812022499634e-08,1.90670246805125e-08,1.45809601283191e-10,-5.79952016893026e-11,-1.31801213491786,655315786.683502,27622325.5059154,1002.15583473466,152.123694477124,4.68235771287718,-0.879421224520134,0.295557179902801,0.154554140362405,-0.0229156709130378,-0.0120515386613554,0.000607446604243751,0.000414778418822002,-7.95490500916542e-06,-7.38526360172807e-06,5.20166719010377e-08,6.65088818539687e-08,-1.35772438545797e-10,-2.39003680063133e-10,0.232108743197644,1051724257.96058,-555976712.570572,966.921596960327,145.469874866832,5.38569112061659,-0.362657959250205,0.127278406047961,0.0780367174408041,-0.00912816258741799,-0.00649145104799418,6.38020463138445e-05,0.000208599818042935,3.16870648396509e-06,-3.3502543800673e-06,-6.08523193986765e-08,2.69791130766542e-08,3.10723693776471e-10,-8.6925527152614e-11,2.31081400221492,246203932.697706,-1336652466.48251,937.453626869778,140.865716663901,6.15039598273493,0.0903840262814978,-0.104376367492142,-0.0122748968832022,0.0123679934086359,0.000790914298733749,-0.000854816316652482,-7.78022259174136e-05,2.27627159134403e-05,2.45173215130342e-06,-2.63126909525082e-07,-3.09808433812687e-08,1.11423084241101e-09,1.38406793314993e-10,-0.926681637845038,-1035372023.47827,533217736.552844,903.869529668514,135.280364451434,4.45827752098917,0.0547545734181628,0.208289010172569,0.0221855672261737,-0.0136158624325514,-0.00272044191824509,0.000212922684389208,7.87088112661446e-05,4.5137323252341e-07,-9.63961918569927e-07,-3.59781059130283e-08,4.74617920035074e-09,2.2137786038681e-10,-4.62471182040111e-12,0.0965858428618496,-223371216.67996,-613694859.379519,872.187197348149,132.685315777722,5.38746308336933,-0.0537108344759256,0.00663811890903925,0.0141154790345001,0.00190121744019454,-0.00127501443267847,-0.000360523434145797,1.0895842413534e-05,1.14456331829487e-05,4.916449113132e-07,-1.41024189287849e-07,-1.0088111514205e-08,6.15688861582362e-10,5.33784839957624e-11,0.738878217908506,-381703875.966159,-378903985.370803,844.826030954265,131.017163797035,4.41918108624226,-0.724842869945408,0.189491244733452,0.114700012802833,-0.0136358493744781,-0.00840994281246125,0.000276849074253616,0.00027335008875125,-1.81474261217307e-06,-4.61543763493164e-06,-6.37751336231016e-09,3.96097044034745e-08,8.70241019854152e-11,-1.36385876777673e-10,0.822430099386811,-446999943.440919,1223252305.40658,814.840919318146,124.68616840001,4.84470935866506,0.0909196853583817,0.0899251640306851,0.00644325859347615,-0.0041247623951232,-0.000977321930567397,-0.000143906328758757,2.97293620416984e-06,7.3997753021468e-06,6.31310237445368e-07,-1.03278890072331e-07,-1.14631238958487e-08,4.7676023644127e-10,5.88736606625339e-11,-0.305378131740878,275700989.466205,-1285250693.06709,788.46109552834,121.472495011351,5.17887046170269,-0.105451890555901,-0.0243502104268151,0.0270120608526967,0.00430487335166178,-0.00213848258933639,-0.000415552907853092,4.44358246801884e-05,1.17586110217271e-05,-2.2256951688079e-07,-1.37346052649981e-07,-2.50657850474402e-09,5.79802573215497e-10,2.22155718821133e-11,0.0368239982086337,-200568420.134781,-209863681.169066,763.509622314375,117.944964843821,5.03672259331534,-0.00551651023103053,-0.0127339727062759,0.0118423923551117,0.00255675032961884,-0.0012349389012175,-0.00031841384173286,1.86582343664266e-05,9.43346781481999e-06,1.66383190397421e-07,-1.12127244314487e-07,-5.52469114318666e-09,4.77802219164745e-10,3.17541437982918e-11,-0.00875069159509952,-274265440.851675,-511636283.849107,739.031357908209,114.637192429481,4.59926490960806,-0.0806449993786145,0.0474126810866465,0.0237184761482357,-0.00125466159664842,-0.0018985572937867,-0.000200222136902156,3.72133171085204e-05,7.58119002731862e-06,-1.00960198474802e-07,-9.81213437149123e-08,-3.66220889993048e-09,4.37578551814315e-10,2.69083483477208e-11,0.373352018626408,-463785508.594968,-224934544.292362,715.509732812743,112.35967170213,4.58860689677725,-0.278108369322017,-0.0201452842709882,0.0365080608530688,0.0052267017207563,-0.00221805927324969,-0.000447357029448433,4.13354024336174e-05,1.2174211046945e-05,-1.49015723553153e-07,-1.39588897316882e-07,-3.06264397664399e-09,5.83285485509742e-10,2.35294188364822e-11,0.552324144243591,-449107891.016072,-240309312.588576,692.374958238243,109.559199804101,4.46572795251365,-0.365653372610769,0.00578828311837584,0.0541902248553733,0.00267892146533822,-0.00354177570781573,-0.000343723245582371,8.88425919336215e-05,1.01465128568752e-05,-1.02701100719285e-06,-1.20455480588358e-07,5.01660536401756e-09,5.13243415492094e-10,-5.77378876883215e-12,0.016122581177518,-963995974.825233,497889297.358085,669.983680217938,105.728920325043,4.15333891379477,-0.279720401033162,0.0571069551867154,0.0477108300047875,-0.0015691905754788,-0.00322799311853759,-0.000170338520980206,8.14023923193653e-05,6.56846485456481e-06,-9.40051524638552e-07,-8.45577543841558e-08,4.55073300775793e-09,3.74195854648304e-10,-4.94200807929336e-12,-0.73571017627664,2089495680.21112,-695533277.810466,649.081875331534,103.975723312709,4.32461818159598,-0.425612899539435,-0.0115026783472369,0.0530667255509518,0.00414786198683875,-0.00301924684712604,-0.000387457091870166,6.33732852645668e-05,1.08013524671434e-05,-4.84897723332907e-07,-1.25537976951271e-07,-4.49209730075482e-10,5.29711118901209e-10,1.54594839399587e-11], aCurrents_HEMS_DH10 := [-9,-8,-7,-6,-5,-4,-3,-2,-1,0.0,1.0,2.0,3.0,4.0,5.0,6.0,7.0,8.0,9.0], aForce_to_current_coefficients_HEMS_DH10 := [1.0,1.0,-7677414494.82291,68609559.3450906,4192502760.98432,-1883602559.27317,247834982.313511,467007.559880945,10016335.7258841,-6167564.21308198,1316507.74565279,-129527.965298496,2955.63053664816,757.118540157646,-100.830512170679,6.39883301415657,-0.243127882295795,0.00563202903490603,-7.36284094309361e-05,4.17624492157816e-07,1.0,1.0,1.0,-652981994.513722,102266852.782046,-64086654.5941818,209278486.002325,-100903517.245318,992945.409165793,13575567.7846208,-5451138.02416426,1151293.36154431,-155248.806495877,14271.500423898,-915.394243537274,40.9811866039206,-1.25502668340294,0.0250470502164369,-0.000293351164098012,1.52865650282461e-06,1.0,1.0,-4620101.20194744,-216338107.495494,-82207401.8385556,-89802509.2112909,138617829.835941,14755834.0638818,-65991322.6267852,35791508.6476587,-10291897.5920975,1887374.09370119,-235548.13095829,20635.670677851,-1281.81391369643,56.119736007193,-1.69146440271729,0.0333675419152579,-0.00038745989813171,2.00611488778097e-06,1.0,-1.97984815540186,-65202310989.8764,56205815148.1442,-15777951426.8194,806395836.481961,203269544.487125,59441137.6524716,-27353387.7431086,777828.390272536,1034182.7824086,-225706.410113207,23297.9145011617,-1287.39718431114,27.2221421858615,1.08059424751822,-0.0960368302854182,0.00301945838939934,-4.66007543184103e-05,2.93554417208605e-07,1.0,1.0,1.0,-521957397.563073,-71363842.7481534,-125737323.964621,357452491.033209,-161194876.902432,-43403.0347846596,21953780.2612293,-8680477.01463083,1821453.83327437,-244391.28948017,22354.7989784959,-1425.83485115375,63.4188499104437,-1.92785356844561,0.038161978821187,-0.000443048988731686,2.28755853615455e-06,1.0,1.0,1.0,-1057161161.55663,-356158716.842664,-70967199.8221605,913480508.658701,-661540064.944938,209628504.631428,-30807848.4103584,-4235.75680898237,863243.281740712,-174112.485853533,19202.4610081049,-1369.6729922441,65.7824974253633,-2.11830637918289,0.0439042776485987,-0.00052960294466283,2.82579530752876e-06,1.0,1.0,1.0,1.0,-2885646112.60472,8332456.36557325,1859736419.07385,-845634027.157113,-978558.024091073,109463858.565857,-42236441.3146657,8685999.44977853,-1150303.16069736,104385.633649191,-6633.24771613561,294.99363962375,-8.99210486905563,0.178889120455141,-0.00209069162623149,1.08793043405637e-05,1.0,1.0,1.0,-5307080.83151688,14645055.2239934,6829042.10030972,201850186.528085,-241297542.379012,120099322.19841,-33108477.243754,5527747.06015964,-553251.53999151,28643.5861843078,199.688029092371,-146.788388507172,11.2326915262458,-0.45850457135249,0.011021535187426,-0.00014726448593167,8.46668735822482e-07,1.0,1.0,1.0,1.0,-17051765968.7626,-138806010.75115,20673465504.9594,-18026689046.009,7847176875.4024,-2136110274.29961,395904068.667885,-52089464.898358,4972189.42030274,-347317.425919693,17720.9687142908,-651.883702979547,16.8078311354812,-0.287826070951925,0.00293689268949705,-1.35007630816887e-05,1.0,1.0,811549046.710949,-149475485.440848,-1291275893.61991,-10362415.0331029,199764541.606793,464059376.6712,-498990653.882176,222669954.187012,-58520094.3240599,10129460.9326803,-1212332.75259614,102787.545674958,-6217.28062597961,266.293510154384,-7.88114053380176,0.153128866675246,-0.00175578213466637,8.99573250838259e-06,1.0,1.0,1.0,1.0,-3371050218.00404,-490943253.987793,4698292545.39979,-3880316526.49424,1621173364.86254,-420077690.943893,72867328.384087,-8741336.1807156,733808.247729859,-42660.3193401471,1652.86566210275,-38.3576892802183,0.329675368650977,0.00697375343446397,-0.000212767418567771,1.68439338434569e-06,1.0,1.0,1.0,1.0,1.0,-25846215509.891,39001760536.4664,-26379343819.405,10585676358.3409,-2812421979.08354,522864997.261601,-70097449.2229781,6884644.77221464,-497853.061314808,26395.6794203264,-1011.15361921383,27.1778020689649,-0.48531169513381,0.00516280670545619,-2.47311582126345e-05,1.0,1.0,-6406978663.67101,-206947748.824033,-509573078.529337,-90504639.3396987,2144843179.6801,-1693437011.85491,566832692.299253,-86985060.3766225,160407.270411104,2524238.52751059,-523339.569572753,59012.2617839461,-4291.87804772301,209.720436487576,-6.8570385729823,0.144015920416231,-0.0017570033440034,9.46421055539376e-06,1.0,1.0,1.0,1.0,-1200297872.54093,138297594.540753,17908916.4206913,591107471.943408,-575271933.360964,256130260.834524,-68352410.7020867,12074872.8258458,-1475947.14538559,127692.337673762,-7866.23981891187,342.280349826855,-10.2629529246932,0.201467925916912,-0.0023278187501352,1.19896171939419e-05,1.0,1.0,1.0,-7841644261.901,3121200511.29756,-1053689.36997665,563057853.486974,-408373712.972993,-3617963.22360008,76318900.2151761,-31912068.0674432,6985901.67994996,-970225.693583778,91460.5039097272,-5994.92024360401,273.474659515798,-8.51244124685207,0.172285787926687,-0.00204212436559241,1.07496115834754e-05,1.0,1.0,-32740431533.9167,15438144175.4194,-456596465.552448,-1488146397.90048,1744207374.92295,-1061945851.15834,269807686.763739,395653.147291995,-18051290.8610798,5296837.00691397,-832822.618564586,84277.1063913065,-5787.41525907369,272.894040439124,-8.70717264155904,0.179634740094364,-0.00216187204005599,1.15211584195052e-05,1.0,1.0,1.0,1.0,-936443043.662185,-19298994.3513026,-37394.9253824199,630356337.058914,-589984366.581241,259439548.01118,-69031456.8572148,12218188.7401196,-1500597.06055004,130707.08222985,-8117.87199602191,356.456600283999,-10.7922844710141,0.21400356102348,-0.00249812087007692,1.2999692692305e-05,-3675561460.63155,1364478865.62357,-645821423.539382,-4700985314.49093,-77256957.1611427,-122576473.842627,2599956655.24841,-1977929254.16465,638684239.098029,-93520141.5240369,-696311.656569201,2854430.38986413,-569311.939720207,62769.4261180864,-4486.08717169224,215.990876887835,-6.97142278394795,0.144759540065463,-0.00174837392706699,9.33427873693846e-06,1.0,1.0,1.0,1.0,-2924132516.39986,-177287740.617338,2601727743.97267,-1586850042.87644,366510265.55779,229966.683614703,-21050837.711128,5891819.81797252,-893037.043884704,87808.4339610303,-5893.23181843465,272.773878650319,-8.5718222441452,0.174621580265185,-0.0020793962427981,1.09828501955125e-05], fK_D_pit := 0, fK_D_roll := 0, fK_D_tot := 0, fK_F_init_pit := 0, fK_F_init_roll := 0, fK_F_init_tot := 0, fK_F_pit := 0, fK_F_roll := 0, fK_F_tot := 0, fK_I_init_pit := 0, fK_I_init_roll := 0, fK_I_init_tot := 0, fK_I_pit := 0, fK_I_roll := 0, fK_I_tot := 0, fK_P_pit := 0, fK_P_roll := 0, fK_P_tot := 0, fd_HEMS_to_HEMS := 0.314, fenable_extra_roll_notch := 1, ff_extra_roll_filter := 652, fg := 9.811999999999999, flift_off_time := 5, fm := 1780, fnotch_damp := 0.3, fnotch_gmin := 0.1, fpitch_target := 0, ar_motor_left_com := [0.0147302,0.8070598,0.34816], ar_motor_right_com := [0.0147302,-0.7979402,0.34816], ar_pitch_hems := [0.8879802,0.8879802,0.8585198,0.8585198], ar_roll_hems := [0.3785598,0.3694402,0.3785598,0.3694402], froll_target := 0, fz_initial_lift_off := -0.023, fz_manual_target := -0.016, fz_mismatch_D := 0, fz_mismatch_F := 100, fz_mismatch_I := 0.0001, fz_mismatch_P := 0.001, bfeed_forward_ems_ON := FALSE, bfeed_fwd_motor_roll_ON := FALSE, blevi_operational := FALSE, blift_off_enabled := TRUE, bmismatch_enabled := FALSE, amismatch_specific_enabler := [FALSE,FALSE,FALSE], bpitch_ON := TRUE, broll_ON := TRUE, broll_filter_enabled := TRUE, btotal_ON := TRUE, fDiscreteDerivative_ICPrevScaledInput := 0, fPIDController_InitialConditionForFilter := 0, fPIDController_InitialConditionForFilter_a := 0, fPIDController_InitialConditionForFilter_j := 0, fPIDController_InitialConditionForIntegrator := 1, fPIDController_InitialConditionForIntegrator_m := 1, fPIDController_InitialConditionForIntegrator_p := 1, fPIDController_LowerSaturationLimit := 0, fPIDController_LowerSaturationLimit_n := 0, fPIDController_LowerSaturationLimit_e := 0, fPIDController_UpperSaturationLimit := 5, fPIDController_UpperSaturationLimit_n := 5, fPIDController_UpperSaturationLimit_g := 5, fConstant1_Value := 0, fConstant1_Value_b := 0, fConstant1_Value_e := 0, fConstant4_Value := 9, fConstant4_Value_e := 0, fUnitDelay_InitialCondition := 0, fIntegrator1_IC := 0, fConstant5_Value := 1, fSwitch1_Threshold := 7, fConstant7_Value := 4.5, fSwitch1_Threshold_i := 0, fsat_enabled_Value := 1, fConstant8_Value := -9, fConstant9_Value := -4.5, fSwitch2_Threshold := 0, fDelay_InitialCondition := 0, fUnitDelay1_InitialCondition := 0, fConstant_Value := 1, fstop_div_by_zero_Threshold := 0, ferror_integrator_IC := 0, ftime_integrator_IC := 0, fConstant_Value_c := 318.3061676617178, ftau_Gain := 0.00075, fBias_Bias := 1, ftwo_Gain := 2, fone_Gain := 1, fUnitDelay1_InitialCondition_m := 0, fTSamp_WtEt := 666.6666666666666, fGain_Gain := -1, ff_roll_n_Value := 318.3061676617178, ftau_Gain_h := 0.00075, fBias_Bias_j := 1, fdamp_roll_notch_Value := 0.3, ftwo_Gain_h := 2, fg_roll_notch_Value := 0.1, fone_Gain_l := 1, fUnitDelay1_InitialCondition_h := 0, ftau_Gain_b := 0.00075, fBias_Bias_c := 1, ftwo_Gain_f := 2, fone_Gain_g := 1, fUnitDelay1_InitialCondition_c := 0, fSwitch_Threshold := 0, fGain1_Gain := -1, ftau_Gain_d := 0.00075, fBias_Bias_g := 1, ftwo_Gain_fc := 2, fone_Gain_f := 1, fUnitDelay1_InitialCondition_ci := 0, fdist_enabled_Value := 1, fUnitDelay1_InitialCondition_n := 0, fConstant_Value_e := 1, fstop_div_by_zero_Threshold_g := 0, fUnitDelay1_InitialCondition_nc := 0, fConstant_Value_a := 1, fstop_div_by_zero_Threshold_p := 0, fZeroGain_Gain := 0, fZeroGain_Gain_m := 0, fZeroGain_Gain_a := 0, fConstant_Value_o := 1, fBias1_Bias := 1, fGain_Gain_p := 2, fUnitDelay2_InitialCondition := 0, fBias1_Bias_d := 1, fGain_Gain_c := 2, fUnitDelay2_InitialCondition_j := 0, fBias1_Bias_l := 1, fGain_Gain_d := 2, fUnitDelay2_InitialCondition_p := 0, fBias1_Bias_j := 1, fGain_Gain_a := 2, fUnitDelay2_InitialCondition_a := 0, fConstant10_Value := 1, fConstant6_Value := 1, fConstant7_Value_o := 0, fConstant8_Value_h := 1, fConstant9_Value_p := 0, fIntegrator2_IC := 0, fIsPeak1_Threshold := 4.5, fSwitch2_Threshold_n := 7, fConstant2_Value := 0, fConstant2_Value_e := 0, fConstant2_Value_d := 0, fDelay1_InitialCondition := 0, fwasfmenabledlastrun_Threshold := 0, fhard_disable_fmm_Gain := 0, fusefmornot_Threshold := 0, bMemory_InitialCondition := FALSE, bMemory_InitialCondition_m := FALSE, bMemory_InitialCondition_n := FALSE, nSwitch_Threshold_c := 0);
	END_STRUCT
END_TYPE

// DUTs/ST_FB_vertical_levitation_control_TcCOM_InitStruct_FB_init
{attribute 'TcIecLibraryType'}
{attribute 'hide'}
TYPE ST_FB_vertical_levitation_control_TcCOM_InitStruct_FB_init : 
	STRUCT
		{attribute 'GUID' := '18071995-0000-0000-0000-000000000018'}
		pInst : PVOID;
		bInitRetains : BOOL;
		bInCopyCode : BOOL;
		 {attribute 'hide'}
		_reserved1 : UINT_16_48;
		stInit : REFERENCE TO ST_FB_vertical_levitation_control_TcCOM_InitStruct;
		result : BOOL;
		 {attribute 'hide'}
		_reserved2 : UINT_24_56;
	END_STRUCT
END_TYPE

// DUTs/ST_FB_vertical_levitation_control_TcCOM_InitStruct_FB_afterinit
{attribute 'TcIecLibraryType'}
{attribute 'hide'}
TYPE ST_FB_vertical_levitation_control_TcCOM_InitStruct_FB_afterinit : 
	STRUCT
		{attribute 'GUID' := '18071995-0000-0000-0000-000000000018'}
		pInst : PVOID;
		result : BOOL;
		 {attribute 'hide'}
		_reserved1 : UINT_24_56;
	END_STRUCT
END_TYPE

// DUTs/ST_FB_vertical_levitation_control_TcCOM_InitStruct_Reinit
{attribute 'TcIecLibraryType'}
{attribute 'hide'}
TYPE ST_FB_vertical_levitation_control_TcCOM_InitStruct_Reinit : 
	STRUCT
		{attribute 'GUID' := '18071995-0000-0000-0000-000000000018'}
		pInst : PVOID;
		stReInit : ST_FB_vertical_levitation_control_TcCOM_InitStruct;
		result : BOOL;
		 {attribute 'hide'}
		_reserved1 : ARRAY [1..7] OF USINT;
	END_STRUCT
END_TYPE

// DUTs/ST_FB_vertical_levitation_control_TcCOM_InitStruct_FB_Main
{attribute 'TcIecLibraryType'}
{attribute 'hide'}
TYPE ST_FB_vertical_levitation_control_TcCOM_InitStruct_FB_Main : 
	STRUCT
		{attribute 'GUID' := '18071995-0000-0000-0000-000000000018'}
		pInst : PVOID;
		result : BOOL;
		 {attribute 'hide'}
		_reserved1 : UINT_24_56;
	END_STRUCT
END_TYPE

// DUTs/ST_FB_vertical_levitation_control_TcCOM_InitStruct_FB_exit
{attribute 'TcIecLibraryType'}
{attribute 'hide'}
TYPE ST_FB_vertical_levitation_control_TcCOM_InitStruct_FB_exit : 
	STRUCT
		{attribute 'GUID' := '18071995-0000-0000-0000-000000000018'}
		pInst : PVOID;
		bInCopyCode : BOOL;
		result : BOOL;
		 {attribute 'hide'}
		_reserved1 : UINT_16_48;
	END_STRUCT
END_TYPE

// DUTs/ST_GetSet_TCOM_STATE
{attribute 'TcIecLibraryType'}
{attribute 'hide'}
TYPE ST_GetSet_TCOM_STATE : 
	STRUCT
		{attribute 'GUID' := '18071995-0000-0000-0000-000000000018'}
		pInst : PVOID;
		{attribute 'GUID' := '18071995-0000-0000-0000-000000000061'}
		eParam : TCOM_STATE;
		 {attribute 'hide'}
		_reserved1 : UINT_0_32;
	END_STRUCT
END_TYPE

// DUTs/ST_GetSet_ITComObject
{attribute 'TcIecLibraryType'}
{attribute 'hide'}
TYPE ST_GetSet_ITComObject : 
	STRUCT
		{attribute 'GUID' := '18071995-0000-0000-0000-000000000018'}
		pInst : PVOID;
		{attribute 'GUID' := '00000012-0000-0000-E000-000000000064'}
		ipParam : ITComObject;
	END_STRUCT
END_TYPE

// DUTs/ST_GetSet_ITcADI
{attribute 'TcIecLibraryType'}
{attribute 'hide'}
TYPE ST_GetSet_ITcADI : 
	STRUCT
		{attribute 'GUID' := '18071995-0000-0000-0000-000000000018'}
		pInst : PVOID;
		{attribute 'GUID' := '03000012-0000-0000-E000-000000000064'}
		ipParam : ITcADI;
	END_STRUCT
END_TYPE

// DUTs/ST_vertical_levitation_control_U_T
(* Generated from type 'vertical_levitation_control_U_T' *)
{attribute 'TcIecLibraryType'}
TYPE ST_vertical_levitation_control_U_T : 
	STRUCT
		(* Generated from item 'z_avg' *)
		fz_avg : LREAL;
		(* Generated from item 'roll_measured' *)
		froll_measured : LREAL;
		(* Generated from item 'pitch_measured' *)
		fpitch_measured : LREAL;
		(* Generated from item 'ems_roll' *)
		fems_roll : LREAL;
		(* Generated from item 'F_imu' *)
		aF_imu : T_matrix3xdouble;
		(* Generated from item 'gyro_imu' *)
		agyro_imu : T_matrix3xdouble;
		(* Generated from item 'motor_Fy_l' *)
		fmotor_Fy_l : LREAL;
		(* Generated from item 'motor_Fy_r' *)
		fmotor_Fy_r : LREAL;
		(* Generated from item 'Feedback_current_hems' *)
		fFeedback_current_hems : LREAL;
	END_STRUCT
END_TYPE

// DUTs/ST_vertical_levitation_control_Y_T
(* Generated from type 'vertical_levitation_control_Y_T' *)
{attribute 'TcIecLibraryType'}
TYPE ST_vertical_levitation_control_Y_T : 
	STRUCT
		(* Generated from item 'I_VFL' *)
		aI_VFL : T_matrix2xdouble;
		(* Generated from item 'I_VFR' *)
		aI_VFR : T_matrix2xdouble;
		(* Generated from item 'I_VBL' *)
		aI_VBL : T_matrix2xdouble;
		(* Generated from item 'I_VBR' *)
		aI_VBR : T_matrix2xdouble;
		(* Generated from item 'F_hems' *)
		aF_hems : T_matrix4xdouble;
		(* Generated from item 'F_requested' *)
		aF_requested : T_matrix3xdouble;
		(* Generated from item 'integral_terms' *)
		aintegral_terms : T_matrix3xdouble;
		(* Generated from item 'sat_failed' *)
		fsat_failed : LREAL;
		(* Generated from item 'net_post_sat' *)
		anet_post_sat : T_matrix3xdouble;
		(* Generated from item 'z_target_adjusted' *)
		fz_target_adjusted : LREAL;
		(* Generated from item 'Max_allowed_current' *)
		aMax_allowed_current : T_matrix4xdouble;
		(* Generated from item 'Min_allowed_current' *)
		aMin_allowed_current : T_matrix4xdouble;
		(* Generated from item 'Avg_total_hems_current' *)
		fAvg_total_hems_current : LREAL;
		(* Generated from item 'Avg_current_hems' *)
		fAvg_current_hems : LREAL;
	END_STRUCT
END_TYPE

